// TwinCAT 3 PLC project PLC1
// ProgramVersion: 3.1.4024.12
// libraries:
//   Tc2_Standard, * (Beckhoff Automation GmbH)
//   Tc2_System, * (Beckhoff Automation GmbH)
//   Tc3_Module, * (Beckhoff Automation GmbH)
//   TcUnit,1.2.0.0,www.tcunit.org
// project tree:
//   GVLs/ GVL.TcGVL
//   / PlcTask.TcTTO
//   POUs/Casts/ CastHelper.TcPOU
//   POUs/Delegate/ Action_I_Observer_.TcPOU, Action_Person_.TcPOU, I_Action.TcIO, I_Predicate.TcIO, Predicate_Person_.TcPOU
//   POUs/ I_Equatable.TcIO, I_Observer.TcIO, Tests.TcPOU, Object.TcPOU, Person.TcPOU, PropertyObserver.TcPOU
//   POUs/List/ List.TcPOU, List_I_Observer_.TcPOU, List_Person_.TcPOU, List_Person_Test.TcPOU, List_I_Observer_Test.TcPOU

CONFIGURATION PLC1
    RESOURCE PLC ON TwinCAT3
        TASK PlcTask(INTERVAL := T#10ms, PRIORITY := 20);
        PROGRAM Tests WITH PlcTask : Tests;
    END_RESOURCE
END_CONFIGURATION

// ---- GVLs/GVL.TcGVL
{attribute 'qualified_only'}
VAR_GLOBAL
    CastHelper : CastHelper;
END_VAR
VAR_GLOBAL CONSTANT
    LIST_UPPER_BOUND : INT := 9;
END_VAR

// ---- POUs/Delegate/I_Action.TcIO
(*
Encapsulates a Perform method that has two parameters and does not return a value
*)
INTERFACE I_Action

(*
Purpose: Encapsulates several methods that can be used in the ForEach loop of a List through all elements.
Since Generic is not supported in Tc you need to implement one FB of your desired type (Action_X_) if you want to use "ForEach" method of a List that needs an Action as an input.
Because you might need several actions for different situations, it's better to write a switch-case statement and put each action in one Case instead of creating multiple FBs.
Later you can pass the CaseNumber to call your desired action.
Parameters: performCaseNumber:INT, Number to choose between actions in the method; item:POINTER TO Object, The object that is passed by the List and can be used in actions.
*)
METHOD Perform
VAR_INPUT
    performCaseNumber : INT;
END_VAR
VAR_IN_OUT
    item : POINTER TO Object;
END_VAR
END_METHOD

END_INTERFACE

// ---- POUs/Delegate/I_Predicate.TcIO
(*
Represents the Evaluate method that defines a set of criteria and determines whether the specified object meets one of those criteria
*)
INTERFACE I_Predicate

(*
Purpose: Defines a set of criteria and determines whether the specified object meets one of those criteria. 
Since Generic is not supported in Tc you need to implement one FB of your desired type (Predicated_X_) if you want to use methods of a List that need Predicate as an input.
Because you might need several criterias for different situations, it's better to write a switch-case statement and put each criteria in one Case instead of creating multiple FBs.
Later you can pass the CaseNumber to call your desired criteria.
Parameters: evaluateCaseNumber:INT, Number to choose between criterias in the method; item:POINTER TO Object, The object to compare against the criteria defined within one of the casees in the method.
Return: BOOL, True if item meets the criteria defined within the method, otherwise False.
*)
METHOD Evaluate : BOOL
VAR_INPUT
    evaluateCaseNumber : INT;
END_VAR
VAR_IN_OUT
    item : POINTER TO Object;
END_VAR
END_METHOD

END_INTERFACE

// ---- POUs/I_Equatable.TcIO
INTERFACE I_Equatable EXTENDS __System.IQueryInterface

METHOD Equals : BOOL
VAR_INPUT
    other : I_Equatable;
END_VAR
END_METHOD

END_INTERFACE

// ---- POUs/I_Observer.TcIO
INTERFACE I_Observer EXTENDS __SYSTEM.IQueryInterface, I_Equatable

METHOD OnError
VAR_INPUT
END_VAR
END_METHOD

METHOD OnUpdate
VAR_INPUT
END_VAR
END_METHOD

END_INTERFACE

// ---- POUs/Tests.TcPOU
PROGRAM Tests
VAR
    list_Person_Test : List_Person_Test;
    list_I_Observer_Test : List_I_Observer_Test;
END_VAR

TcUnit.RUN();

END_PROGRAM

// ---- POUs/List/List_Person_Test.TcPOU
FUNCTION_BLOCK List_Person_Test EXTENDS TcUnit.FB_TestSuite

AddItem();
AddRange();
Clear();
Contains();
Exists();
Find();
FindAll();
FindIndex();
FindLast();
FindLastIndex();
Foreach();
GetCapacity();
GetCount();
GetItem();
GetRange();
IndexOfItem();
LastIndexOfItem();
Initialize();
Insert();
InsertRange();
Remove();
RemoveAll();
RemoveAt();
RemoveRange();

METHOD AddItem
VAR
    personsList : List_Person_;
    personA : Person;
    personB : Person;
    actualIndex1 : INT;
    actualIndex2 : INT;
    j : INT;
END_VAR
TEST('AddPersonShouldReturnAddedIndex');
//Assign
//Act
actualIndex1 := personsList.AddItem(personA);
actualIndex2 := personsList.AddItem(personB);
//Assert
AssertEquals_INT(0, actualIndex1,'check add 1');
AssertEquals_INT(1, actualIndex2,'check add 2');
TEST_FINISHED();

TEST('AddToAFullListShouldReturnMinusOne');
//Assign
personsList.Clear();
FOR j:=0 TO GVL.LIST_UPPER_BOUND DO
    personsList.AddItem(personA);
END_FOR
//Act
actualIndex1 := personsList.AddItem(personB);
//Assert
AssertEquals_INT(-1, actualIndex1,'check overflow add');
TEST_FINISHED();
END_METHOD

METHOD AddRange
VAR
    personsList : List_Person_;
    personA : Person;
    personB : Person;
    personC : Person;
    personD : Person;
    personE : Person;
    personF : Person;
    personG : Person;
    validArrayPtPerson : ARRAY[0..2] OF POINTER TO Person := [ADR(personE), ADR(personF), ADR(personG)];
    unvalidArrayPtPerson : ARRAY[0..6 + 1] OF POINTER TO Person;
    actualPtPerson3 : POINTER TO Person;
    actualPtPerson4 : POINTER TO Person;
    actualPtPerson5 : POINTER TO Person;
    actualPtPerson6 : POINTER TO Person;
    expected : INT := 6;
    actual : INT;
END_VAR
//Before All
personA.SetAge(10);
personB.SetAge(11);
personC.SetAge(12);
personD.SetAge(13);
personE.SetAge(14);
personF.SetAge(15);
personG.SetAge(16);
personA.SetName('A');
personB.SetName('B');
personC.SetName('C');
personD.SetName('D');
personE.SetName('E');
personF.SetName('F');
personG.SetName('G');

TEST('AddRangeShouldPassAndReturnTheLastIndex');
//Assign
personsList.AddItem(personA);
personsList.AddItem(personB);
personsList.AddItem(personC);
personsList.AddItem(personD);
//Act
actual := personsList.AddRange(validArrayPtPerson);
actualPtPerson3 := personsList.GetItem(3);
actualPtPerson4 := personsList.GetItem(4);
actualPtPerson5 := personsList.GetItem(5);
actualPtPerson6 := personsList.GetItem(6);
//Assert
AssertEquals(expected, actual, 'check result');
AssertEquals_INT(7, personsList.GetCount(),'check list count');
AssertTrue(actualPtPerson3^.Equals(personD),'check added element 3');
AssertTrue(actualPtPerson4^.Equals(personE),'check added element 4');
AssertTrue(actualPtPerson5^.Equals(personF),'check added element 5');
AssertTrue(actualPtPerson6^.Equals(personG),'check added element 6');
TEST_FINISHED();

TEST('AddRangeShouldFailAndReturnMinusOne');
//Assign
personsList.Clear();
personsList.AddItem(personA);
personsList.AddItem(personB);
personsList.AddItem(personC);
personsList.AddItem(personD);
expected := -1;
//Act
actual := personsList.AddRange(unvalidArrayPtPerson);
//Assert
AssertEquals(expected, actual, 'check result');
AssertEquals_INT(4, personsList.GetCount(),'check list count');
TEST_FINISHED();
END_METHOD

METHOD Clear
VAR
    personsList1 : List_Person_;
    personsList2 : List_Person_;
    person : Person;
    expectedCount : INT := 0;
    actualCount : INT;
END_VAR
TEST('ClearAFilledListShouldPass');
//Assign
personsList1.AddItem(person);
//Act
personsList1.Clear();
actualCount := personsList1.GetCount();
//Assert
AssertEquals(expectedCount, actualCount,'');
TEST_FINISHED();

TEST('ClearAnEmptyListShouldPass');
//Assign
expectedCount := 0;
//Act
personsList2.Clear();
actualCount := personsList2.GetCount();
//Assert
AssertEquals(expectedCount, actualCount,'');
TEST_FINISHED();
END_METHOD

METHOD Contains
VAR
    personsList : List_Person_;
    personA : Person;
    personB : Person;
    personC : Person;
    personD : Person;
    personE : Person;
    personF : Person;
    personG : Person;
    actual : BOOL;
END_VAR
//Before All
personA.SetAge(10);
personB.SetAge(11);
personC.SetAge(12);
personD.SetAge(13);
personE.SetAge(14);
personF.SetAge(15);
personG.SetAge(16);
personA.SetName('A');
personB.SetName('B');
personC.SetName('C');
personD.SetName('D');
personE.SetName('E');
personF.SetName('F');
personG.SetName('G');
personsList.AddItem(personA);
personsList.AddItem(personB);
personsList.AddItem(personC);
personsList.AddItem(personD);
personsList.AddItem(personE);
personsList.AddItem(personF);

TEST('ContainsShouldReturnTrue');
//Assign
//Act
actual := personsList.Contains(personC);
//Assert
AssertTrue(actual,'Looking for personC');
TEST_FINISHED();

TEST('ContainsShouldReturnFalse');
//Assign
//Act
actual := personsList.Contains(personG);
//Assert
AssertFalse(actual,'Looking for personG');
TEST_FINISHED();
END_METHOD

METHOD Exists
VAR
    personsList : List_Person_;
    personA : Person;
    personB : Person;
    personC : Person;
    personD : Person;
    personE : Person;
    personF : Person;
    personG : Person;
    predicate_Person_ : Predicate_Person_;
    actual : BOOL;
END_VAR
//Before All
personA.SetAge(10);
personB.SetAge(11);
personC.SetAge(12);
personD.SetAge(13);
personE.SetAge(14);
personF.SetAge(15);
personG.SetAge(16);
personA.SetName('A');
personB.SetName('B');
personC.SetName('C');
personD.SetName('D');
personE.SetName('E');
personF.SetName('F');
personG.SetName('G');
personsList.AddItem(personA);
personsList.AddItem(personB);
personsList.AddItem(personC);
personsList.AddItem(personD);
personsList.AddItem(personE);
personsList.AddItem(personF);

TEST('ExistsShouldReturnTrue');
//Assign
//Act
actual := personsList.Exists(predicate_Person_, 2);
//Assert
AssertTrue(actual,'Looking for a person with name C');
TEST_FINISHED();

TEST('ExistsShouldReturnFalse');
//Assign
//Act
actual := personsList.Exists(predicate_Person_, 3);
//Assert
AssertFalse(actual,'Looking for a person with name G');
TEST_FINISHED();
END_METHOD

METHOD Find
VAR
    personsList : List_Person_;
    personA : Person;
    personB : Person;
    personC : Person;
    personD : Person;
    personE : Person;
    personF : Person;
    personG : Person;
    predicate_Person_ : Predicate_Person_;
    actualPtPerson : POINTER TO Person;
    nullPtPerson : POINTER TO person := 0;
END_VAR
//Before All
personA.SetAge(10);
personB.SetAge(11);
personC.SetAge(12);
personD.SetAge(13);
personE.SetAge(14);
personF.SetAge(15);
personG.SetAge(16);
personA.SetName('A');
personB.SetName('B');
personC.SetName('C');
personD.SetName('D');
personE.SetName('E');
personF.SetName('F');
personG.SetName('G');
personsList.AddItem(personA);
personsList.AddItem(personB);
personsList.AddItem(personC);
personsList.AddItem(personD);
personsList.AddItem(personE);
personsList.AddItem(personF);

TEST('FindShouldReturnAPerson');
//Assign
//Act
actualPtPerson := personsList.Find(predicate_Person_, 2);
//Assert
AssertTrue(actualPtPerson^.Equals(personC),'Get person with name C');
TEST_FINISHED();

TEST('FindShouldReturnZero');
//Assign
//Act
actualPtPerson := personsList.Find(predicate_Person_, 3);
//Assert
AssertEquals(nullPtPerson, actualPtPerson,'Get Zero when looking for person with name G');
TEST_FINISHED();
END_METHOD

METHOD FindAll
VAR
    personsList : List_Person_;
    personA : Person;
    personB : Person;
    personC : Person;
    personD : Person;
    personE : Person;
    personF : Person;
    predicate_Person_ : Predicate_Person_;
    actualPersonsList : list_Person_;
    actualCount : INT;
    expectedCount : INT := 3;
    actualPtPerson0 : POINTER TO Person;
    actualPtPerson1 : POINTER TO Person;
    actualPtPerson2 : POINTER TO Person;
    nullPtPerson : POINTER TO Person := 0;
END_VAR
//Before All
personA.SetAge(10);
personB.SetAge(11);
personC.SetAge(12);
personD.SetAge(13);
personE.SetAge(14);
personF.SetAge(15);
personsList.AddItem(personA);
personsList.AddItem(personB);
personsList.AddItem(personC);
personsList.AddItem(personD);
personsList.AddItem(personE);
personsList.AddItem(personF);

TEST('FindAllShouldReturnAProperList');
//Assign
//Act
actualPersonsList := personsList.FindAll(predicate_Person_, 1); //Get people younger than 13
actualCount := actualPersonsList.GetCount();
actualPtPerson0 := actualPersonsList.GetItem(0);
actualPtPerson1 := actualPersonsList.GetItem(1);
actualPtPerson2 := actualPersonsList.GetItem(2);
//Assert
AssertEquals(expectedCount, actualCount, 'Check new list count');
AssertTrue(actualPtPerson0^.Equals(personA),'First element should personA');
AssertTrue(actualPtPerson1^.Equals(personB),'First element should personB');
AssertTrue(actualPtPerson2^.Equals(personC),'First element should personC');
TEST_FINISHED();

TEST('FindAllShouldReturnAnEmptyList');
//Assign
expectedCount := 0;
//Act
actualPersonsList := personsList.FindAll(predicate_Person_, 4); //Get people older than 50
actualCount := actualPersonsList.GetCount();
actualPtPerson0 := actualPersonsList.GetItem(0);
//Assert
AssertEquals(expectedCount, actualCount, 'Check new list count');
AssertEquals(nullPtPerson, actualPtPerson0, 'Check returned list element 0');
TEST_FINISHED();
END_METHOD

METHOD FindIndex
VAR
    personsList : List_Person_;
    personA : Person;
    personB : Person;
    personC : Person;
    personD : Person;
    personE : Person;
    personF : Person;
    personG : Person;
    predicate_Person_ : Predicate_Person_;
    actualIndex : INT;
    expectedIndex : INT := 2;
END_VAR
//Before All
personA.SetAge(10);
personB.SetAge(11);
personC.SetAge(12);
personD.SetAge(13);
personE.SetAge(14);
personF.SetAge(15);
personG.SetAge(16);
personA.SetName('A');
personB.SetName('B');
personC.SetName('C');
personD.SetName('D');
personE.SetName('E');
personF.SetName('F');
personG.SetName('G');
personsList.AddItem(personA);
personsList.AddItem(personB);
personsList.AddItem(personC);
personsList.AddItem(personD);
personsList.AddItem(personE);
personsList.AddItem(personF);

TEST('FindIndexShouldReturnTheIndex');
//Assign
//Act
actualIndex := personsList.FindIndex(predicate_Person_, 2);
//Assert
AssertEquals(expectedIndex, actualIndex, 'find person with name C index');
TEST_FINISHED();

TEST('FindIndexShouldReturnMinusOne');
//Assign
expectedIndex := -1;
//Act
actualIndex := personsList.FindIndex(predicate_Person_, 3);
//Assert
AssertEquals(expectedIndex, actualIndex, 'Find person with name G index');
TEST_FINISHED();
END_METHOD

METHOD FindLast
VAR
    personsList : List_Person_;
    personA : Person;
    personB : Person;
    personC : Person;
    personC2 : Person;
    personD : Person;
    personE : Person;
    personF : Person;
    personG : Person;
    predicate_Person_ : Predicate_Person_;
    actualPtPerson : POINTER TO Person;
    nullPtPerson : POINTER TO person := 0;
END_VAR
//Before All
personA.SetAge(10);
personB.SetAge(11);
personC.SetAge(12);
personC2.SetAge(22);
personD.SetAge(13);
personE.SetAge(14);
personF.SetAge(15);
personG.SetAge(16);
personA.SetName('A');
personB.SetName('B');
personC.SetName('C');
personC2.SetName('C');
personD.SetName('D');
personE.SetName('E');
personF.SetName('F');
personG.SetName('G');
personsList.AddItem(personA);
personsList.AddItem(personB);
personsList.AddItem(personC);
personsList.AddItem(personD);
personsList.AddItem(personE);
personsList.AddItem(personC2); //Duplicated C
personsList.AddItem(personF);

TEST('FindLastShouldReturnAPerson');
//Assign
//Act
actualPtPerson := personsList.FindLast(predicate_Person_, 2);
//Assert
AssertFalse(actualPtPerson^.Equals(personC),'Not the last person with name C');
AssertTrue(actualPtPerson^.Equals(personC2),'Be the last person with name C');
TEST_FINISHED();

TEST('FindLastShouldReturnNull');
//Assign
//Act
actualPtPerson := personsList.Find(predicate_Person_, 3);
//Assert
AssertEquals(nullPtPerson, actualPtPerson,'Get Zero when looking for person with name G');
TEST_FINISHED();
END_METHOD

METHOD FindLastIndex
VAR
    personsList : List_Person_;
    personA : Person;
    personB : Person;
    personC : Person;
    personC2 : Person;
    personD : Person;
    personE : Person;
    personF : Person;
    personG : Person;
    predicate_Person_ : Predicate_Person_;
    actualIndex : INT;
    expectedIndex : INT := 5;
END_VAR
//Before All
personA.SetAge(10);
personB.SetAge(11);
personC.SetAge(12);
personC.SetAge(22);
personD.SetAge(13);
personE.SetAge(14);
personF.SetAge(15);
personG.SetAge(16);
personA.SetName('A');
personB.SetName('B');
personC.SetName('C');
personC2.SetName('C');
personD.SetName('D');
personE.SetName('E');
personF.SetName('F');
personG.SetName('G');
personsList.AddItem(personA);
personsList.AddItem(personB);
personsList.AddItem(personC);
personsList.AddItem(personD);
personsList.AddItem(personE);
personsList.AddItem(personC2);
personsList.AddItem(personF);

TEST('FindLastIndexShouldReturnTheIndex');
//Assign
//Act
actualIndex := personsList.FindLastIndex(predicate_Person_, 2);
//Assert
AssertEquals(expectedIndex, actualIndex, 'Find last person with name C index');
TEST_FINISHED();

TEST('FindLastIndexShouldReturnMinusOne');
//Assign
expectedIndex := -1;
//Act
actualIndex := personsList.FindLastIndex(predicate_Person_, 3);
//Assert
AssertEquals(expectedIndex, actualIndex, 'Find person with name G index');
TEST_FINISHED();
END_METHOD

METHOD Foreach
VAR
    personsList : List_Person_;
    personA : Person;
    personB : Person;
    personC : Person;
    personD : Person;
    personE : Person;
    personF : Person;
    personG : Person;
    action_Person_ : Action_Person_;
    actualPtPersonArray : ARRAY[0..3] OF POINTER TO Person;
    j : INT;
    expectedName : STRING := 'John';
END_VAR
TEST('ForeachShouldPass');
//Assign
personA.SetAge(10);
personB.SetAge(11);
personC.SetAge(12);
personD.SetAge(13);
personE.SetAge(14);
personF.SetAge(15);
personG.SetAge(16);
personA.SetName('A');
personB.SetName('B');
personC.SetName('C');
personD.SetName('D');
personE.SetName('E');
personF.SetName('F');
personG.SetName('G');
personsList.AddItem(personA);
personsList.AddItem(personB);
personsList.AddItem(personC);
personsList.AddItem(personD);
//Act
personsList.Foreach(action_Person_, 2);
FOR j:=0 TO 3 DO
    actualPtPersonArray[j] := personsList.GetItem(j);
END_FOR
//Assert
AssertEquals_STRING(expectedName, actualPtPersonArray[0]^.GetName(),'element 0 shuold be named John');
AssertEquals_STRING(expectedName, actualPtPersonArray[1]^.GetName(),'element 0 shuold be named John');
AssertEquals_STRING(expectedName, actualPtPersonArray[2]^.GetName(),'element 0 shuold be named John');
AssertEquals_STRING(expectedName, actualPtPersonArray[3]^.GetName(),'element 0 shuold be named John');
TEST_FINISHED();
END_METHOD

METHOD GetCapacity
VAR
    personsList : List_Person_;
    person : Person;
    expectedCapacity : INT := GVL.LIST_UPPER_BOUND + 1;
    actualCapacity : INT;
END_VAR
TEST('GetCapacityShouldPass');
//Act
actualCapacity := personsList.GetCapacity();
//Assert
AssertEquals_INT(expectedCapacity, actualCapacity,'Get capacity at the begining');
TEST_FINISHED();

TEST('GetCapacityShouldPassWithSameValue');
//Assign
personsList.AddItem(person);
//Act
actualCapacity := personsList.GetCapacity();
//Assert
AssertEquals(expectedCapacity, actualCapacity,'Get capacity after adding a person');
TEST_FINISHED();
END_METHOD

METHOD GetCount
VAR
    personsList : List_Person_;
    person : Person;
    expectedCount : INT := 0;
    actualCount : INT;
END_VAR
TEST('GetCountShouldReturnZero');
//Act
actualCount := personsList.GetCount();
//Assert
AssertEquals_INT(expectedCount, actualCount,'Get count at the begining');
TEST_FINISHED();

TEST('GetCountShouldReturnOne');
//Assign
personsList.AddItem(person);
expectedCount := 1;
//Act
actualCount := personsList.GetCount();
//Assert
AssertEquals(expectedCount, actualCount,'Get count after adding a person');
TEST_FINISHED();
END_METHOD

METHOD GetItem
VAR
    personsList : List_Person_;
    personA : Person;
    personB : Person;
    actualPtPerson : POINTER TO Person;
END_VAR
//Before All
personA.SetAge(10);
personB.SetAge(11);
personA.SetName('A');
personB.SetName('B');
personsList.AddItem(personA);
personsList.AddItem(personB);

TEST('GetPersonShouldPass');
//Assign
//Act
actualPtPerson := personsList.GetItem(1);
//Assert
AssertEquals_INT(11, actualPtPerson^.GetAge(),'check age');
AssertTrue(actualPtPerson^.Equals(personB),'check Equality');
TEST_FINISHED();

TEST('GetShouldBeByReference');
//Assign
//Act
actualPtPerson := personsList.GetItem(1);
personB.SetAge(20);
actualPtPerson^.GetAge();
//Assert
AssertEquals_INT(20, actualPtPerson^.GetAge(),'');
TEST_FINISHED();
END_METHOD

METHOD GetRange
VAR
    personsList : List_Person_;
    personA : Person;
    personB : Person;
    personC : Person;
    personD : Person;
    personE : Person;
    personF : Person;
    personG : Person;
    actualPersonsList : list_Person_;
    actualCount : INT;
    expectedCount : INT := 3;
    actualPtPerson0 : POINTER TO Person;
    actualPtPerson1 : POINTER TO Person;
    actualPtPerson2 : POINTER TO Person;
END_VAR
//Before All
personA.SetAge(10);
personB.SetAge(11);
personC.SetAge(12);
personD.SetAge(13);
personE.SetAge(14);
personF.SetAge(15);
personG.SetAge(16);
personsList.AddItem(personA);
personsList.AddItem(personB);
personsList.AddItem(personC);
personsList.AddItem(personD);
personsList.AddItem(personE);
personsList.AddItem(personF);

TEST('GetRangeShouldReturnList');
//Assign
//Act
actualPersonsList := personsList.GetRange(1, expectedCount);
actualCount := actualPersonsList.GetCount();
actualPtPerson0 := actualPersonsList.GetItem(0);
actualPtPerson1 := actualPersonsList.GetItem(1);
actualPtPerson2 := actualPersonsList.GetItem(2);
//Assert
AssertEquals(expectedCount, actualCount, 'Check new list count');
AssertTrue(actualPtPerson0^.Equals(personB),'First element should personB');
AssertTrue(actualPtPerson1^.Equals(personC),'First element should personC');
AssertTrue(actualPtPerson2^.Equals(personD),'First element should personD');
TEST_FINISHED();

TEST('GetRangeShouldReturnListTillLastElement');
//Assign
//Act
actualPersonsList := personsList.GetRange(1, 1000);
actualCount := actualPersonsList.GetCount();
//Assert
expectedCount := 5;
AssertEquals(expectedCount, actualCount, 'Check new list count for GetRange 1000');
TEST_FINISHED();

TEST('GetRangeShouldReturnEmptyList');
//Assign
//Act
actualPersonsList := personsList.GetRange(-5, 1);
actualCount := actualPersonsList.GetCount();
//Assert
expectedCount := 0;
AssertEquals(expectedCount, actualCount, 'Check new list count for GetRange starting -5');
TEST_FINISHED();
END_METHOD

METHOD IndexOfItem
VAR
    personsList : List_Person_;
    personA : Person;
    personB : Person;
    personC : Person;
    personD : Person;
    personE : Person;
    personF : Person;
    personG : Person;
    actualIndex : INT;
    expectedIndex : INT := 3;
END_VAR
//Before All
personA.SetAge(10);
personB.SetAge(11);
personC.SetAge(12);
personD.SetAge(13);
personE.SetAge(14);
personF.SetAge(15);
personG.SetAge(16);
personA.SetName('A');
personB.SetName('B');
personC.SetName('C');
personD.SetName('D');
personE.SetName('E');
personF.SetName('F');
personG.SetName('G');
personsList.AddItem(personA);
personsList.AddItem(personB);
personsList.AddItem(personC);
personsList.AddItem(personD);
personsList.AddItem(personE);
personsList.AddItem(personF);

TEST('IndexOfItemShouldReturnTheIndex');
//Assign
//Act
actualIndex := personsList.IndexOfItem(personD);
//Assert
AssertEquals(expectedIndex, actualIndex, 'return the index of personD');
TEST_FINISHED();

TEST('IndexOfItemShouldReturnMinusOne');
//Assign
//Act
actualIndex := personsList.IndexOfItem(personG);
//Assert
expectedIndex := -1;
AssertEquals(expectedIndex, actualIndex, 'return the index of personG');
TEST_FINISHED();
END_METHOD

METHOD Initialize
VAR
    personsList : List_Person_;
    personA : Person;
    personB : Person;
    personC : Person;
    validArrayPtPerson : ARRAY[0..2] OF POINTER TO Person := [ADR(personA), ADR(personB), ADR(personC)];
    unvalidArrayPtPerson : ARRAY[0..GVL.LIST_UPPER_BOUND + 1] OF POINTER TO Person;
    actualPtPerson0 : POINTER TO Person;
    actualPtPerson1 : POINTER TO Person;
    actualPtPerson2 : POINTER TO Person;
    expected : INT := 2;
    actual : INT;
END_VAR
//Before All
personA.SetAge(10);
personB.SetAge(11);
personC.SetAge(12);
personA.SetName('A');
personB.SetName('B');
personC.SetName('C');

TEST('InitializeShouldPassAndReturnTheLastIndex');
//Assign
//Act
actual := personsList.Initialize(validArrayPtPerson);
actualPtPerson0 := personsList.GetItem(0);
actualPtPerson1 := personsList.GetItem(1);
actualPtPerson2 := personsList.GetItem(2);
//Assert
AssertEquals(expected, actual, 'check result');
AssertEquals_INT(3, personsList.GetCount(),'check list count');
AssertTrue(actualPtPerson0^.Equals(personA),'check added element 0');
AssertTrue(actualPtPerson1^.Equals(personB),'check added element 1');
AssertTrue(actualPtPerson2^.Equals(personC),'check added element 2');
TEST_FINISHED();

TEST('InitializeShouldFailAndReturnMinusOne');
//Assign
personsList.Clear();
expected := -1;
//Act
actual := personsList.Initialize(unvalidArrayPtPerson);
//Assert
AssertEquals(expected, actual, 'check result');
AssertEquals_INT(0, personsList.GetCount(),'check list count');
TEST_FINISHED();
END_METHOD

METHOD Insert
VAR
    personsList : List_Person_;
    personA : Person;
    personB : Person;
    personC : Person;
    personD : Person;
    actualPtPerson1 : POINTER TO Person;
    actualPtPerson2 : POINTER TO Person;
    actualPtPerson3 : POINTER TO Person;
    expected : INT := 2;
    actual : INT;
END_VAR
//Before All
personA.SetAge(10);
personB.SetAge(11);
personC.SetAge(12);
personD.SetAge(13);
personA.SetName('A');
personB.SetName('B');
personC.SetName('C');
personD.SetName('D');

TEST('InsertShouldPassAndReturnTheLastIndex');
//Assign
personsList.AddItem(personA);
personsList.AddItem(personB);
personsList.AddItem(personC);
//Act
actual := personsList.Insert(2, personD);
actualPtPerson1 := personsList.GetItem(1);
actualPtPerson2 := personsList.GetItem(2);
actualPtPerson3 := personsList.GetItem(3);
//Assert
AssertEquals(expected, actual, 'check result');
AssertEquals_INT(4, personsList.GetCount(),'check list count');
AssertTrue(actualPtPerson1^.Equals(personB),'check added element 1');
AssertTrue(actualPtPerson2^.Equals(personD),'check added element 2');
AssertTrue(actualPtPerson3^.Equals(personC),'check added element 3');
TEST_FINISHED();

TEST('InsertShouldPassEvenByIndexHigherThanListCurrentLastIndexAndReturnTheLastIndex');
//Assign
personsList.Clear();
personsList.AddItem(personA);
personsList.AddItem(personB);
personsList.AddItem(personC);
expected := 3;
//Act
actual := personsList.Insert(7, personD);
actualPtPerson1 := personsList.GetItem(1);
actualPtPerson2 := personsList.GetItem(2);
actualPtPerson3 := personsList.GetItem(3);
//Assert
AssertEquals(expected, actual, 'check result');
AssertEquals_INT(4, personsList.GetCount(),'check list count');
AssertTrue(actualPtPerson1^.Equals(personB),'check added element 1');
AssertTrue(actualPtPerson2^.Equals(personC),'check added element 2');
AssertTrue(actualPtPerson3^.Equals(personD),'check added element 3');
TEST_FINISHED();

TEST('InsertShouldPassEvenByIndexHigherThanListUpperBoundAndReturnTheLastIndex');
//Assign
personsList.Clear();
personsList.AddItem(personA);
personsList.AddItem(personB);
personsList.AddItem(personC);
expected := 3;
//Act
actual := personsList.Insert(GVL.LIST_UPPER_BOUND + 1, personD);
actualPtPerson1 := personsList.GetItem(1);
actualPtPerson2 := personsList.GetItem(2);
actualPtPerson3 := personsList.GetItem(3);
//Assert
AssertEquals(expected, actual, 'check result');
AssertEquals_INT(4, personsList.GetCount(),'check list count');
AssertTrue(actualPtPerson1^.Equals(personB),'check added element 1');
AssertTrue(actualPtPerson2^.Equals(personC),'check added element 2');
AssertTrue(actualPtPerson3^.Equals(personD),'check added element 3');
TEST_FINISHED();

TEST('InsertShouldFailByMinusIndexAndReturnMinusOne');
//Assign
personsList.Clear();
personsList.AddItem(personA);
personsList.AddItem(personB);
personsList.AddItem(personC);
expected := -1;
//Act
actual := personsList.Insert(-1, personD);
//Assert
AssertEquals(expected, actual, 'check result');
AssertEquals_INT(3, personsList.GetCount(),'check list count');
TEST_FINISHED();
END_METHOD

METHOD InsertRange
VAR
    personsList : List_Person_;
    personA : Person;
    personB : Person;
    personC : Person;
    personD : Person;
    personE : Person;
    personF : Person;
    personG : Person;
    validArrayPtPerson : ARRAY[0..2] OF POINTER TO Person := [ADR(personE), ADR(personF), ADR(personG)];
    unvalidArrayPtPerson : ARRAY[0..6 + 1] OF POINTER TO Person;
    actualPtPerson1 : POINTER TO Person;
    actualPtPerson2 : POINTER TO Person;
    actualPtPerson3 : POINTER TO Person;
    actualPtPerson4 : POINTER TO Person;
    actualPtPerson5 : POINTER TO Person;
    actualPtPerson6 : POINTER TO Person;
    actualPtPerson7 : POINTER TO Person;
    expected : INT := 4;
    actual : INT;
END_VAR
//Before All
personA.SetAge(10);
personB.SetAge(11);
personC.SetAge(12);
personD.SetAge(13);
personE.SetAge(14);
personF.SetAge(15);
personG.SetAge(16);
personA.SetName('A');
personB.SetName('B');
personC.SetName('C');
personD.SetName('D');
personE.SetName('E');
personF.SetName('F');
personG.SetName('G');

TEST('InsertRangeShouldPassAndReturnTheLastIndex');
//Assign
personsList.AddItem(personA);
personsList.AddItem(personB);
personsList.AddItem(personC);
personsList.AddItem(personD);
//Act
actual := personsList.InsertRange(2, validArrayPtPerson);
actualPtPerson1 := personsList.GetItem(1);
actualPtPerson2 := personsList.GetItem(2);
actualPtPerson3 := personsList.GetItem(3);
actualPtPerson4 := personsList.GetItem(4);
actualPtPerson5 := personsList.GetItem(5);
//Assert
AssertEquals(expected, actual, 'check result');
AssertEquals_INT(7, personsList.GetCount(),'check list count');
AssertTrue(actualPtPerson1^.Equals(personB),'check added element 1');
AssertTrue(actualPtPerson2^.Equals(personE),'check added element 2');
AssertTrue(actualPtPerson3^.Equals(personF),'check added element 3');
AssertTrue(actualPtPerson4^.Equals(personG),'check added element 4');
AssertTrue(actualPtPerson5^.Equals(personC),'check added element 5');
TEST_FINISHED();

TEST('InsertRangeShouldPassEvenByIndexHigherThanListCurrentLastIndexAndReturnTheLastIndex');
//Assign
personsList.Clear();
personsList.AddItem(personA);
personsList.AddItem(personB);
personsList.AddItem(personC);
personsList.AddItem(personD);
expected := 6;
//Act
actual := personsList.InsertRange(7, validArrayPtPerson);
actualPtPerson3 := personsList.GetItem(3);
actualPtPerson4 := personsList.GetItem(4);
actualPtPerson5 := personsList.GetItem(5);
actualPtPerson6 := personsList.GetItem(6);
//Assert
AssertEquals(expected, actual, 'check result');
AssertEquals_INT(7, personsList.GetCount(),'check list count');
AssertTrue(actualPtPerson3^.Equals(personD),'check added element 3');
AssertTrue(actualPtPerson4^.Equals(personE),'check added element 4');
AssertTrue(actualPtPerson5^.Equals(personF),'check added element 5');
AssertTrue(actualPtPerson6^.Equals(personG),'check added element 6');
TEST_FINISHED();

TEST('InsertRangeShouldPassEvenByIndexHigherThanListUpperBoundAndReturnTheLastIndex');
//Assign
personsList.Clear();
personsList.AddItem(personA);
personsList.AddItem(personB);
personsList.AddItem(personC);
personsList.AddItem(personD);
expected := 6;
//Act
actual := personsList.InsertRange(7, validArrayPtPerson);
actualPtPerson3 := personsList.GetItem(3);
actualPtPerson4 := personsList.GetItem(4);
actualPtPerson5 := personsList.GetItem(5);
actualPtPerson6 := personsList.GetItem(6);
//Assert
AssertEquals(expected, actual, 'check result');
AssertEquals_INT(7, personsList.GetCount(),'check list count');
AssertTrue(actualPtPerson3^.Equals(personD),'check added element 3');
AssertTrue(actualPtPerson4^.Equals(personE),'check added element 4');
AssertTrue(actualPtPerson5^.Equals(personF),'check added element 5');
AssertTrue(actualPtPerson6^.Equals(personG),'check added element 6');
TEST_FINISHED();

TEST('InsertRangeShouldFailByMinusIndexAndReturnMinusOne');
//Assign
personsList.Clear();
personsList.AddItem(personA);
personsList.AddItem(personB);
personsList.AddItem(personC);
personsList.AddItem(personD);
expected := -1;
//Act
actual := personsList.InsertRange(-1, validArrayPtPerson);
//Assert
AssertEquals(expected, actual, 'check result');
AssertEquals_INT(4, personsList.GetCount(),'check list count');
TEST_FINISHED();

TEST('InsertRangeShouldFailByLongArrayLengthAndReturnMinusOne');
//Assign
personsList.Clear();
personsList.AddItem(personA);
personsList.AddItem(personB);
personsList.AddItem(personC);
personsList.AddItem(personD);
expected := -1;
//Act
actual := personsList.InsertRange(2, unvalidArrayPtPerson);
//Assert
AssertEquals(expected, actual, 'check result');
AssertEquals_INT(4, personsList.GetCount(),'check list count');
TEST_FINISHED();
END_METHOD

METHOD LastIndexOfItem
VAR
    personsList : List_Person_;
    personA : Person;
    personB : Person;
    personC : Person;
    personD : Person;
    personE : Person;
    personF : Person;
    personG : Person;
    actualIndex : INT;
    expectedIndex : INT := 5;
END_VAR
//Before All
personA.SetAge(10);
personB.SetAge(11);
personC.SetAge(12);
personD.SetAge(13);
personE.SetAge(14);
personF.SetAge(15);
personG.SetAge(16);
personA.SetName('A');
personB.SetName('B');
personC.SetName('C');
personD.SetName('D');
personE.SetName('E');
personF.SetName('F');
personG.SetName('G');
personsList.AddItem(personA);
personsList.AddItem(personB);
personsList.AddItem(personC);
personsList.AddItem(personD);
personsList.AddItem(personE);
personsList.AddItem(personD);
personsList.AddItem(personF);

TEST('LastIndexOfItemShouldReturnTheIndex');
//Assign
//Act
actualIndex := personsList.LastIndexOfItem(personD);
//Assert
AssertEquals(expectedIndex, actualIndex, 'return the last index of personD');
TEST_FINISHED();

TEST('LastIndexOfItemShouldReturnMinusOne');
//Assign
//Act
actualIndex := personsList.LastIndexOfItem(personG);
//Assert
expectedIndex := -1;
AssertEquals(expectedIndex, actualIndex, 'return the last index of personG');
TEST_FINISHED();
END_METHOD

METHOD Remove
VAR
    personsList : List_Person_;
    personA : Person;
    personB : Person;
    personC : Person;
    personD : Person;
    expectedCount : INT := 3;
    actualPtPerson1 : POINTER TO Person;
    actualPtPerson2 : POINTER TO Person;
    actualCount : INT;
    actual : BOOL;
END_VAR
//Before All
personA.SetAge(10);
personB.SetAge(11);
personC.SetAge(12);
personD.SetAge(13);
personA.SetName('A');
personB.SetName('B');
personC.SetName('C');
personD.SetName('D');
personsList.AddItem(personA);
personsList.AddItem(personB);
personsList.AddItem(personC);
personsList.AddItem(personD);

TEST('RemoveShouldPassAndReturnTrue');
//Assign
//Act
actual := personsList.Remove(personC);
actualCount := personsList.GetCount();
actualPtPerson1 := personsList.GetItem(1);
actualPtPerson2 := personsList.GetItem(2);
//Assert
AssertTrue(actual,'check result of remove');
AssertEquals(expectedCount, actualCount,'check list count');
AssertTrue(actualPtPerson1^.Equals(personB),'check list element 1');
AssertTrue(actualPtPerson2^.Equals(personD),'check list element 2');
TEST_FINISHED();

TEST('RemoveShouldFailAndReturnFalse');
//Assign
//Act
actual := personsList.Remove(personC);
actualCount := personsList.GetCount();
actualPtPerson1 := personsList.GetItem(1);
actualPtPerson2 := personsList.GetItem(2);
//Assert
AssertFalse(actual,'check result of remove');
AssertEquals(expectedCount, actualCount,'check list count');
AssertTrue(actualPtPerson1^.Equals(personB),'check list element 1');
AssertTrue(actualPtPerson2^.Equals(personD),'check list element 2');
TEST_FINISHED();
END_METHOD

METHOD RemoveAll
VAR
    personsList : List_Person_;
    personA : Person;
    personB : Person;
    personC : Person;
    personD : Person;
    personE : Person;
    personF : Person;
    personG : Person;
    predicate_Person_ : Predicate_Person_;
    actual : INT;
    expected : INT := 3;
    actualCount : INT;
    expectedCount : INT := 4;
    actualPtPerson0 : POINTER TO Person;
    actualPtPerson1 : POINTER TO Person;
    actualPtPerson2 : POINTER TO Person;
    actualPtPerson3 : POINTER TO Person;
    actualPtPerson4 : POINTER TO Person;
    actualPtPerson5 : POINTER TO Person;
    actualPtPerson6 : POINTER TO Person;
END_VAR
//Before All
personA.SetAge(10);
personB.SetAge(11);
personC.SetAge(12);
personD.SetAge(13);
personE.SetAge(14);
personF.SetAge(15);
personG.SetAge(16);

TEST('RemoveAllShouldReturnAProperList');
//Assign
personsList.AddItem(personA);
personsList.AddItem(personB);
personsList.AddItem(personC);
personsList.AddItem(personD);
personsList.AddItem(personE);
personsList.AddItem(personF);
personsList.AddItem(personG);
//Act
actual := personsList.RemoveAll(predicate_Person_, 1); //Remove people younger than 13
actualCount := personsList.GetCount();
actualPtPerson0 := personsList.GetItem(0);
actualPtPerson1 := personsList.GetItem(1);
actualPtPerson2 := personsList.GetItem(2);
actualPtPerson3 := personsList.GetItem(3);
//Assert
AssertEquals(expected, actual, 'check result');
AssertEquals(expectedCount, actualCount, 'check list count');
AssertTrue(actualPtPerson0^.Equals(personD),'check returned list element 0');
AssertTrue(actualPtPerson1^.Equals(personE),'check returned list element 1');
AssertTrue(actualPtPerson2^.Equals(personF),'check returned list element 2');
AssertTrue(actualPtPerson3^.Equals(personG),'check returned list element 3');
TEST_FINISHED();

TEST('RemoveAllShouldReturnTheOriginalListUntouched');
//Assign
personsList.Clear();
personsList.AddItem(personA);
personsList.AddItem(personB);
personsList.AddItem(personC);
personsList.AddItem(personD);
personsList.AddItem(personE);
personsList.AddItem(personF);
personsList.AddItem(personG);
expected := 0;
expectedCount := 7;
//Act
actual := personsList.RemoveAll(predicate_Person_, 4); //Remove people older than 50
actualCount := personsList.GetCount();
actualPtPerson0 := personsList.GetItem(0);
actualPtPerson1 := personsList.GetItem(1);
actualPtPerson2 := personsList.GetItem(2);
actualPtPerson3 := personsList.GetItem(3);
actualPtPerson4 := personsList.GetItem(4);
actualPtPerson5 := personsList.GetItem(5);
actualPtPerson6 := personsList.GetItem(6);
//Assert
AssertEquals(expected, actual, 'check result');
AssertEquals(expectedCount, actualCount, 'check list count');
AssertTrue(actualPtPerson0^.Equals(personA),'check returned list element 0');
AssertTrue(actualPtPerson1^.Equals(personB),'check returned list element 1');
AssertTrue(actualPtPerson2^.Equals(personC),'check returned list element 2');
AssertTrue(actualPtPerson3^.Equals(personD),'check returned list element 3');
AssertTrue(actualPtPerson4^.Equals(personE),'check returned list element 4');
AssertTrue(actualPtPerson5^.Equals(personF),'check returned list element 5');
AssertTrue(actualPtPerson6^.Equals(personG),'check returned list element 6');
TEST_FINISHED();
END_METHOD

METHOD RemoveAt
VAR
    personsList : List_Person_;
    personA : Person;
    personB : Person;
    personC : Person;
    personD : Person;
    actualPtPersonArray : ARRAY[0..3] OF POINTER TO Person;
    expectedCount : INT := 3;
    actualCount : INT;
    actual : BOOL;
    j : INT;
END_VAR
//Before All
personA.SetAge(10);
personB.SetAge(11);
personC.SetAge(12);
personD.SetAge(13);
personA.SetName('A');
personB.SetName('B');
personC.SetName('C');
personD.SetName('D');

TEST('RemoveAtShouldPass');
//Assign
personsList.Clear();
personsList.AddItem(personA);
personsList.AddItem(personB);
personsList.AddItem(personC);
personsList.AddItem(personD);
//Act
actual := personsList.RemoveAt(2);
actualCount := personsList.GetCount();
FOR j:=0 TO 3 DO
    actualPtPersonArray[j] := personsList.GetItem(j);
END_FOR
//Assert
AssertTrue(actual,'check result of remove');
AssertEquals(expectedCount, actualCount,'check list count');
AssertTrue(actualPtPersonArray[0]^.Equals(personA),'check element 0');
AssertTrue(actualPtPersonArray[1]^.Equals(personB),'check element 1');
AssertTrue(actualPtPersonArray[2]^.Equals(personD),'check element 2');
TEST_FINISHED();

TEST('RemoveAtMinusIndexShouldFail');
//Assign
personsList.Clear();
personsList.AddItem(personA);
personsList.AddItem(personB);
personsList.AddItem(personC);
personsList.AddItem(personD);
expectedCount := 4;
//Act
actual := personsList.RemoveAt(-1);
actualCount := personsList.GetCount();
FOR j:=0 TO 3 DO
    actualPtPersonArray[j] := personsList.GetItem(j);
END_FOR
//Assert
AssertFalse(actual,'check result of remove');
AssertEquals(expectedCount, actualCount,'check list count');
AssertTrue(actualPtPersonArray[0]^.Equals(personA),'check element 0');
AssertTrue(actualPtPersonArray[1]^.Equals(personB),'check element 1');
AssertTrue(actualPtPersonArray[2]^.Equals(personC),'check element 2');
AssertTrue(actualPtPersonArray[3]^.Equals(personD),'check element 3');
TEST_FINISHED();

TEST('RemoveAtIndexGreaterThanLastIndexShouldFail');
//Assign
personsList.Clear();
personsList.AddItem(personA);
personsList.AddItem(personB);
personsList.AddItem(personC);
personsList.AddItem(personD);
expectedCount := 4;
//Act
actualCount := personsList.GetCount();
actual := personsList.RemoveAt(actualCount);
actualCount := personsList.GetCount();
FOR j:=0 TO 3 DO
    actualPtPersonArray[j] := personsList.GetItem(j);
END_FOR
//Assert
AssertFalse(actual,'check result of remove');
AssertEquals(expectedCount, actualCount,'check list count');
AssertTrue(actualPtPersonArray[0]^.Equals(personA),'check element 0');
AssertTrue(actualPtPersonArray[1]^.Equals(personB),'check element 1');
AssertTrue(actualPtPersonArray[2]^.Equals(personC),'check element 2');
AssertTrue(actualPtPersonArray[3]^.Equals(personD),'check element 3');
TEST_FINISHED();
END_METHOD

METHOD RemoveRange
VAR
    personsList : List_Person_;
    personA : Person;
    personB : Person;
    personC : Person;
    personD : Person;
    personE : Person;
    personF : Person;
    personG : Person;
    actualPtPersonArray : ARRAY[0..3] OF POINTER TO Person;
    expectedCount : INT := 7 - 3;
    actualCount : INT;
    actual : BOOL;
    j : INT;
END_VAR
//Before All
personA.SetAge(10);
personB.SetAge(11);
personC.SetAge(12);
personD.SetAge(13);
personE.SetAge(14);
personF.SetAge(15);
personG.SetAge(16);
personA.SetName('A');
personB.SetName('B');
personC.SetName('C');
personD.SetName('D');
personE.SetName('E');
personF.SetName('F');
personG.SetName('G');

TEST('RemoveRangeShouldPass');
//Assign
personsList.AddItem(personA);
personsList.AddItem(personB);
personsList.AddItem(personC);
personsList.AddItem(personD);
personsList.AddItem(personE);
personsList.AddItem(personF);
personsList.AddItem(personG);
//Act
actual := personsList.RemoveRange(2,3);
actualCount := personsList.GetCount();
FOR j:=0 TO 3 DO
    actualPtPersonArray[j] := personsList.GetItem(j);
END_FOR
//Assert
AssertTrue(actual,'check result of removeRange');
AssertEquals(expectedCount, actualCount,'check list count');
AssertTrue(actualPtPersonArray[0]^.Equals(personA),'check element 0');
AssertTrue(actualPtPersonArray[1]^.Equals(personB),'check element 1');
AssertTrue(actualPtPersonArray[2]^.Equals(personF),'check element 2');
AssertTrue(actualPtPersonArray[3]^.Equals(personG),'check element 3');
TEST_FINISHED();

TEST('RemoveRangeWithRangeLongerThanCountShouldPass');
//Assign
personsList.Clear();
personsList.AddItem(personA);
personsList.AddItem(personB);
personsList.AddItem(personC);
personsList.AddItem(personD);
personsList.AddItem(personE);
personsList.AddItem(personF);
personsList.AddItem(personG);
expectedCount := 4;
//Act
actual := personsList.RemoveRange(4,10);
actualCount := personsList.GetCount();
FOR j:=0 TO 3 DO
    actualPtPersonArray[j] := personsList.GetItem(j);
END_FOR
//Assert
AssertTrue(actual,'check result of removeRange');
AssertEquals(expectedCount, actualCount,'check list count');
AssertTrue(actualPtPersonArray[0]^.Equals(personA),'check element 0');
AssertTrue(actualPtPersonArray[1]^.Equals(personB),'check element 1');
AssertTrue(actualPtPersonArray[2]^.Equals(personC),'check element 2');
AssertTrue(actualPtPersonArray[3]^.Equals(personD),'check element 3');
TEST_FINISHED();

TEST('RemoveRangeWithMinusIndexShouldFail');
//Assign
personsList.Clear();
personsList.AddItem(personA);
personsList.AddItem(personB);
personsList.AddItem(personC);
personsList.AddItem(personD);
personsList.AddItem(personE);
personsList.AddItem(personF);
personsList.AddItem(personG);
expectedCount := 7;
//Act
actual := personsList.RemoveRange(-1,3);
actualCount := personsList.GetCount();
FOR j:=0 TO 3 DO
    actualPtPersonArray[j] := personsList.GetItem(j);
END_FOR
//Assert
AssertFalse(actual,'check result of removeRange');
AssertEquals(expectedCount, actualCount,'check list count');
AssertTrue(actualPtPersonArray[0]^.Equals(personA),'check element 0');
AssertTrue(actualPtPersonArray[1]^.Equals(personB),'check element 1');
AssertTrue(actualPtPersonArray[2]^.Equals(personC),'check element 2');
AssertTrue(actualPtPersonArray[3]^.Equals(personD),'check element 3');
TEST_FINISHED();

TEST('RemoveRangeWithIndexGreaterThanLastIndexShouldFail');
//Assign
personsList.Clear();
personsList.AddItem(personA);
personsList.AddItem(personB);
personsList.AddItem(personC);
personsList.AddItem(personD);
personsList.AddItem(personE);
personsList.AddItem(personF);
personsList.AddItem(personG);
expectedCount := 7;
//Act
actualCount := personsList.GetCount();
actual := personsList.RemoveRange(actualCount,3);
actualCount := personsList.GetCount();
FOR j:=0 TO 3 DO
    actualPtPersonArray[j] := personsList.GetItem(j);
END_FOR
//Assert
AssertFalse(actual,'check result of removeRange');
AssertEquals(expectedCount, actualCount,'check list count');
AssertTrue(actualPtPersonArray[0]^.Equals(personA),'check element 0');
AssertTrue(actualPtPersonArray[1]^.Equals(personB),'check element 1');
AssertTrue(actualPtPersonArray[2]^.Equals(personC),'check element 2');
AssertTrue(actualPtPersonArray[3]^.Equals(personD),'check element 3');
TEST_FINISHED();
END_METHOD

END_FUNCTION_BLOCK

// ---- POUs/List/List_Person_.TcPOU
(*
Sample List which has all available functionalities.
For instance this is a list of type Person (C# eq: List<Person>).
To have any desired type (!!!Not Interface!!!) make a copy of this FB and change Person to your type in all methods
*)
FUNCTION_BLOCK FINAL List_Person_ EXTENDS List

(*
Purpose: Adds an item to the end of the List
Parameters: item:{X Extends Object}, The object to be added to the end of the List
Return: INT, The zero-based index of added object if item is added, otherwise -1
*)
METHOD PUBLIC AddItem : INT
VAR_IN_OUT
    item : Person;
END_VAR
AddItem := SUPER^._addItem(item);
END_METHOD

(*
Purpose: Adds elements of the specified array to the end of the List
Parameters: items:ARRAY[*] OF POINTER TO {X Extends Object}, The array whose elements should be added to the end of the List
Return: INT, The zero-based index of the last added object if items are added, otherwise -1
*)
METHOD PUBLIC AddRange : INT
VAR_IN_OUT
    items : ARRAY[*] OF POINTER TO Person;
END_VAR
AddRange := SUPER^._addRange(items);
END_METHOD

(*
Purpose: Determines whether an element is in the List
Parameters: item:{X Extends Object}, The object to locate in the List
Return: BOOL, True if item is found in the List, otherwise False
*)
METHOD PUBLIC Contains : BOOL
VAR_IN_OUT
    item: Person;
END_VAR
Contains := SUPER^._contains(item);
END_METHOD

(*
Purpose: Determines whether the List contains elements that match the condition defined by the specified predicate
Parameters: predicate:{Predicate_X_ Implements IPredicate}, The Predicate delegate that defines the conditions of the elements to search for; evaluateCaseNumber:INT, Number that specifies which condition to evaluate
Return: BOOL, True if the List contains one or more elements that match the condition defined by the specified predicate, otherwise False
*)
METHOD PUBLIC Exists : BOOL
VAR_INPUT
    predicate: Predicate_Person_;
    evaluateCaseNumber : INT;
END_VAR
Exists := SUPER^._exists(predicate, evaluateCaseNumber);
END_METHOD

(*
Purpose: Searches for an element that matches the conditions defined by the specified predicate, and returns the first occurrence within the entire List
Parameters: predicate:{Predicate_X_ Implements IPredicate}, The Predicate delegate that defines the conditions of the elements to search for; evaluateCaseNumber:INT, Number that specifies which condition to evaluate
Return: POINTER TO {X Extends Object}, The address of the first element that matches the conditions defined by the specified predicate if found, otherwise 0
*)
METHOD Find : POINTER TO Person
VAR_INPUT
    predicate: Predicate_Person_;
    evaluateCaseNumber : INT;
END_VAR
Find := SUPER^._find(predicate, evaluateCaseNumber);
END_METHOD

(*
Purpose: Retrieves all the elements that match the conditions defined by the specified predicate
Parameters: predicate:{Predicate_X_ Implements IPredicate}, The Predicate delegate that defines the conditions of the elements to search for; evaluateCaseNumber:INT, Number that specifies which condition to evaluate
Return: {List_X_ Extends List}, A List containing all the elements that match the conditions defined by the specified predicate if found, otherwise an empty List
*)
METHOD FindAll: List_Person_
VAR_INPUT
    predicate: Predicate_Person_;
    evaluateCaseNumber : INT;
END_VAR
FindAll := GVL.CastHelper.ListToList_Person_(SUPER^._findAll(predicate, evaluateCaseNumber));
END_METHOD

(*
Purpose: Searches for an element that matches the conditions defined by a specified predicate and returns the zero-based index of the first occurrence within the List
Parameters: predicate:{Predicate_X_ Implements IPredicate}, The Predicate delegate that defines the conditions of the elements to search for; evaluateCaseNumber:INT, Number that specifies which condition to evaluate
Return: INT, The zero-based index of the first occurrence of an element that matches the conditions defined by match if found, otherwise -1.
*)
METHOD FindIndex : INT
VAR_INPUT
    predicate: Predicate_Person_;
    evaluateCaseNumber : INT;
END_VAR
FindIndex := SUPER^._findIndex(predicate, evaluateCaseNumber);
END_METHOD

(*
Purpose: Searches for an element that matches the conditions defined by the specified predicate, and returns the last occurrence within the entire List
Parameters: predicate:{X Implements IPredicate}, The Predicate delegate that defines the conditions of the elements to search for; evaluateCaseNumber:INT, Number that specifies which condition to evaluate
Return: POINTER TO {X Extends Object}, The address of the last element that matches the conditions defined by the specified predicate if found, otherwise 0
*)
METHOD FindLast : POINTER TO Person
VAR_INPUT
    predicate: Predicate_Person_;
    evaluateCaseNumber : INT;
END_VAR
FindLast := SUPER^._findLast(predicate, evaluateCaseNumber);
END_METHOD

(*
Purpose: Searches for an element that matches the conditions defined by a specified predicate and returns the zero-based index of the last occurrence within the List
Parameters: predicate:{X Implements IPredicate}, The Predicate delegate that defines the conditions of the elements to search for; evaluateCaseNumber:INT, Number that specifies which condition to evaluate
Return: INT, The zero-based index of the last occurrence of an element that matches the conditions defined by match if found, otherwise -1.
*)
METHOD FindLastIndex : INT
VAR_INPUT
    predicate: Predicate_Person_;
    evaluateCaseNumber : INT;
END_VAR
FindLastIndex := SUPER^._findLastIndex(predicate, evaluateCaseNumber);
END_METHOD

(*
Purpose: Performs the specified action on each element of the List
Parameters: _action:{Action_X_ Implements IAction}, The Action delegate to perform on each element of the List; performCaseNumber:INT, Number that specifies which action to perform
Return: BOOL, True if the action is performed on all elements, otherwise False
*)
METHOD Foreach: BOOL
VAR_INPUT
    _action : I_Action;
    performCaseNumber : INT;
END_VAR
Foreach := SUPER^._forEach(_action, performCaseNumber);
END_METHOD

(*
Purpose: Gets the element at the specified index
Parameters: index:INT, The zero-based index of the element to get
Return: POINTER TO {X Extends Object}, The element at the specified index
*)
METHOD PUBLIC GetItem : POINTER TO Person
VAR_INPUT
    index : INT;
END_VAR
GetItem := SUPER^.GetItemAsIEquatable(index);
END_METHOD

(*
Purpose: Creates a shallow copy of a range of elements in the source List
Parameters: index:INT, The zero-based List index at which the range starts; count:INT, The number of elements in the range
Return: {List_X_ Extends List}, A shallow copy of a range of elements in the source List
*)
METHOD PUBLIC GetRange: List_Person_
VAR_INPUT
    index : INT;
    count : INT;
END_VAR
GetRange := GVL.CastHelper.ListToList_Person_(SUPER^._getRange(index, count));
END_METHOD

(*
Purpose: Returns the zero-based index of the first occurrence in the List
Parameters: item:{X Extends Object}, The object to locate in the List
Return: INT, The zero-based index of the first occurrence of item in the List if found, otherwise -1
*)
METHOD PUBLIC IndexOfItem : INT
VAR_IN_OUT
    item: Person;
END_VAR
IndexOfItem := SUPER^._indexOf(item);
END_METHOD

(*
Purpose: Initializes the List by copying the specified array
Parameters: items:ARRAY[*] OF POINTER TO {X Extends Object}, The array whose elements are copied to the new list
Return: INT, The zero-based index of the last copied element if input array length is less or equal to length of the list, otherwise -1
*)
METHOD PUBLIC Initialize : INT
VAR_IN_OUT
    items : ARRAY[*] OF POINTER TO Person;
END_VAR
Initialize := _initialize(items);
END_METHOD

(*
Purpose: Inserts an item at the specified index
Parameters: index:INT ,The zero-based index at which the new object should be inserted; item:{X Extends Object}, The object to insert
Return: INT, The zero-based index of the inserted object if inserted, otherwise -1
*)
METHOD PUBLIC Insert : INT
VAR_INPUT
    index : INT;
END_VAR
VAR_IN_OUT
    item : Person;
END_VAR
Insert := SUPER^._insert(index, item);
END_METHOD

(*
Purpose: Inserts elements of the specified array at the specified index
Parameters: index:INT ,The zero-based index at which the new elements should be inserted; items:ARRAY[*] OF POINTER TO {X Extends Object}, The array whose elements should be inserted into the List
Return: INT, The zero-based index of the last inserted object if input array length is less or equal to remaining capacity of the list, otherwise -1
*)
METHOD PUBLIC InsertRange : INT
VAR_INPUT
    index : INT;
END_VAR
VAR_IN_OUT
    items : ARRAY[*] OF POINTER TO Person;
END_VAR
InsertRange := SUPER^._insertRange(index, items);
END_METHOD

(*
Purpose: Returns the zero-based index of the last occurrence in the List
Parameters: item:{X Extends Object}, The object to locate in the List
Return: INT, The zero-based index of the last occurrence of item in the List if found, otherwise -1
*)
METHOD PUBLIC LastIndexOfItem : INT
VAR_IN_OUT
    item: Person;
END_VAR
LastIndexOfItem := SUPER^._lastIndexOf(item);
END_METHOD

(*
Purpose: Removes the address of the first occurrence of a specific object from the List
Parameters: item:{X Extends Object}, The object to remove from the List
Return: BOOL, True if item is successfully removed, otherwise False
*)
METHOD PUBLIC Remove : BOOL
VAR_IN_OUT
    item: Person;
END_VAR
Remove := SUPER^._remove(item);
END_METHOD

(*
Purpose: Removes all the elements that match the conditions defined by the specified predicate
Parameters: predicate:{Predicate_X_ Implements IPredicate}, The Predicate delegate that defines the conditions of the elements to search for; evaluateCaseNumber:INT, Number that specifies which condition to evaluate
Return: INT, The number of elements removed from the List
*)
METHOD RemoveAll : INT
VAR_INPUT
    predicate: Predicate_Person_;
    evaluateCaseNumber : INT;
END_VAR
RemoveAll := SUPER^._removeAll(predicate, evaluateCaseNumber);
END_METHOD

(*
Purpose: Copies the elements of the List to a new array
Return: ARRAY[0..GVL.LIST_UPPER_BOUND] OF POINTER TO {X Extends Object}, An array containing copies of the elements of the List as {X Extends Object}
*)
METHOD PUBLIC ToArray : ARRAY[0..GVL.LIST_UPPER_BOUND] OF POINTER TO Person
VAR
    i : INT;
    arrayOfIEquatable : ARRAY[0..GVL.LIST_UPPER_BOUND] OF POINTER TO I_Equatable;
    _result : ARRAY[0..GVL.LIST_UPPER_BOUND] OF POINTER TO Person;
END_VAR
arrayOfIEquatable := SUPER^._toArray();
FOR i:=0 TO GetCount() - 1 DO
    _result[i] := arrayOfIEquatable[i];
END_FOR

ToArray := _result;
END_METHOD

END_FUNCTION_BLOCK

// ---- POUs/List/List.TcPOU
(*
Base List which includes core and generic functionality of a list.
To have a list of any desired type (X) a new FB that Extends this FB should be created which can implement any desired Protected methods of this FB.
*)
FUNCTION_BLOCK List
VAR_INPUT
END_VAR
VAR_OUTPUT
END_VAR
VAR
    _internalArray : ARRAY [0..GVL.LIST_UPPER_BOUND] OF LWORD;
    _count : INT := 0;
END_VAR

(*
Purpose: Adds the address of an Object to the end of the List
Parameters: item:Object, The object to be added to the end of the List
Return: INT, The zero-based index of added object if item is added, otherwise -1
*)
METHOD PROTECTED _addItem : INT
VAR_IN_OUT
    item : Object;
END_VAR
VAR
    _result : INT := -1;
END_VAR
IF GetCount() <= GVL.LIST_UPPER_BOUND THEN
    _internalArray[_count] := ADR(item);
    _result := _count;
    _count := _count + 1;
END_IF
_addItem := _result;
END_METHOD

(*
Purpose: Adds the address of the elements of the specified array to the end of the List
Parameters: items:ARRAY[*] OF POINTER TO Object, The array whose elements should be added to the end of the List
Return: INT, The zero-based index of the last added object if items are added, otherwise -1
*)
METHOD PROTECTED _addRange : INT
VAR_IN_OUT
    items : ARRAY[*] OF POINTER TO Object;
END_VAR
VAR
    _result : INT := -1;
    _lowerBound : DINT;
    _upperBound : DINT;
    _itemsLength : DINT;
    i : DINT;
END_VAR
_lowerBound := LOWER_BOUND(items,1);
_upperBound := UPPER_BOUND(items,1);
_itemsLength := _upperBound - _lowerBound + 1;
IF _itemsLength <= GetCapacity() - GetCount() THEN
    FOR i := _lowerBound TO _upperBound DO
        _addItem(items[i]^);
	END_FOR
    _result := DINT_TO_INT(GetCount() - 1);
END_IF

_addRange := _result;
END_METHOD

(*
Purpose: Determines whether an element is in the List
Parameters: item:Object, The object to locate in the List
Return: BOOL, True if item is found in the List, otherwise False
*)
METHOD PROTECTED _contains : BOOL
VAR_IN_OUT
    item : Object;
END_VAR
VAR
    i : INT;
    _lastIndex : INT;
    _currentItem : POINTER TO Object;
    _result : BOOL := False;
END_VAR
IF GetCount() > 0 THEN
    _lastIndex := GetCount() - 1;
    FOR i:=0 TO _lastIndex DO
        _currentItem := GetItemAsIEquatable(i);
        IF _currentItem^.Equals(item) THEN
            _result := TRUE;
            EXIT;
        END_IF
    END_FOR
END_IF

_contains := _result;
END_METHOD

(*
Purpose: Determines whether the List contains elements that match the condition defined by the specified predicate
Parameters: predicate:IPredicate, The Predicate delegate that defines the conditions of the elements to search for; evaluateCaseNumber:INT, Number that specifies which condition to evaluate
Return: BOOL, True if the List contains one or more elements that match the condition defined by the specified predicate, otherwise False
*)
METHOD PROTECTED _exists : BOOL
VAR_INPUT
    predicate : I_Predicate;
    evaluateCaseNumber : INT;
END_VAR
VAR
    i : INT;
    _lastIndex : INT;
    _currentItem : POINTER TO Object;
    _result : BOOL := FALSE;
END_VAR
IF GetCount() > 0 THEN
    _lastIndex := GetCount() - 1;
    FOR i:=0 TO _lastIndex DO
        _currentItem := GetItemAsIEquatable(i);
        IF predicate.Evaluate(evaluateCaseNumber, _currentItem) THEN
            _result := TRUE;
            EXIT;
        END_IF
    END_FOR
END_IF

_exists := _result;
END_METHOD

(*
Purpose: Searches for an element that matches the conditions defined by the specified predicate, and returns the first occurrence within the entire List
Parameters: predicate:IPredicate, The Predicate delegate that defines the conditions of the elements to search for; evaluateCaseNumber:INT, Number that specifies which condition to evaluate
Return: POINTER TO Object, The address of the first element that matches the conditions defined by the specified predicate if found, otherwise 0
*)
METHOD PROTECTED _find : POINTER TO Object
VAR_INPUT
    predicate : I_Predicate;
    evaluateCaseNumber : INT;
END_VAR
VAR
    i : INT;
    _lastIndex : INT;
    _currentItem : POINTER TO Object;
    _result : POINTER TO Object := 0;
END_VAR
IF GetCount() > 0 THEN
    _lastIndex := GetCount() - 1;
    FOR i:=0 TO _lastIndex DO
        _currentItem := GetItemAsIEquatable(i);
        IF predicate.Evaluate(evaluateCaseNumber, _currentItem) THEN
            _result := _currentItem;
            EXIT;
        END_IF
    END_FOR
END_IF

_find := _result;
END_METHOD

(*
Purpose: Retrieves all the elements that match the conditions defined by the specified predicate
Parameters: predicate:IPredicate, The Predicate delegate that defines the conditions of the elements to search for; evaluateCaseNumber:INT, Number that specifies which condition to evaluate
Return: List, A List containing all the elements that match the conditions defined by the specified predicate if found, otherwise an empty List
*)
METHOD PROTECTED _findAll : List
VAR_INPUT
    predicate : I_Predicate;
    evaluateCaseNumber : INT;
END_VAR
VAR
    i : INT;
    _lastIndex : INT;
    _currentItem : POINTER TO Object;
    _result : List;
END_VAR
IF GetCount() > 0 THEN
    _lastIndex := GetCount() - 1;
    FOR i:=0 TO _lastIndex DO
        _currentItem := GetItemAsIEquatable(i);
        IF predicate.Evaluate(evaluateCaseNumber, _currentItem) THEN
            _result._addItem(_currentItem^);
        END_IF
    END_FOR
END_IF

_findAll := _result;
END_METHOD

(*
Purpose: Searches for an element that matches the conditions defined by a specified predicate and returns the zero-based index of the first occurrence within the List
Parameters: predicate:IPredicate, The Predicate delegate that defines the conditions of the elements to search for; evaluateCaseNumber:INT, Number that specifies which condition to evaluate
Return: INT, The zero-based index of the first occurrence of an element that matches the conditions defined by match if found, otherwise -1.
*)
METHOD PROTECTED _findIndex : INT
VAR_INPUT
    predicate : I_Predicate;
    evaluateCaseNumber : INT;
END_VAR
VAR
    i : INT;
    _lastIndex : INT;
    _currentItem : POINTER TO Object;
    _result : INT := -1;
END_VAR
IF GetCount() > 0 THEN
    _lastIndex := GetCount() - 1;
    FOR i:=0 TO _lastIndex DO
        _currentItem := GetItemAsIEquatable(i);
        IF predicate.Evaluate(evaluateCaseNumber, _currentItem) THEN
            _result := i;
            EXIT;
        END_IF
    END_FOR
END_IF

_findIndex := _result;
END_METHOD

(*
Purpose: Searches for an element that matches the conditions defined by the specified predicate, and returns the last occurrence within the entire List
Parameters: predicate:IPredicate, The Predicate delegate that defines the conditions of the elements to search for; evaluateCaseNumber:INT, Number that specifies which condition to evaluate
Return: POINTER TO Object, The address of the last element that matches the conditions defined by the specified predicate if found, otherwise 0
*)
METHOD PROTECTED _findLast : POINTER TO Object
VAR_INPUT
    predicate : I_Predicate;
    evaluateCaseNumber : INT;
END_VAR
VAR
    i : INT;
    _lastIndex : INT;
    _currentItem : POINTER TO Object;
    _result : POINTER TO Object := 0;
END_VAR
IF GetCount() > 0 THEN
    _lastIndex := GetCount() - 1;
    FOR i:=0 TO _lastIndex DO
        _currentItem := GetItemAsIEquatable(_lastIndex - i);
        IF predicate.Evaluate(evaluateCaseNumber, _currentItem) THEN
            _result := _currentItem;
            EXIT;
        END_IF
    END_FOR
END_IF

_findLast := _result;
END_METHOD

(*
Purpose: Searches for an element that matches the conditions defined by a specified predicate and returns the zero-based index of the last occurrence within the List
Parameters: predicate:IPredicate, The Predicate delegate that defines the conditions of the elements to search for; evaluateCaseNumber:INT, Number that specifies which condition to evaluate
Return: INT, The zero-based index of the last occurrence of an element that matches the conditions defined by match if found, otherwise -1.
*)
METHOD PROTECTED _findLastIndex : INT
VAR_INPUT
    predicate : I_Predicate;
    evaluateCaseNumber : INT;
END_VAR
VAR
    i : INT;
    _lastIndex : INT;
    _currentItem : POINTER TO Object;
    _result : INT := -1;
END_VAR
IF GetCount() > 0 THEN
    _lastIndex := GetCount() - 1;
    FOR i:=0 TO _lastIndex DO
        _currentItem := GetItemAsIEquatable(_lastIndex - i);
        IF predicate.Evaluate(evaluateCaseNumber, _currentItem) THEN
            _result := _lastIndex - i;
            EXIT;
        END_IF
    END_FOR
END_IF

_findLastIndex := _result;
END_METHOD

(*
Purpose: Performs the specified action on each element of the List
Parameters: _action:IAction, The Action delegate to perform on each element of the List; performCaseNumber:INT, Number that specifies which action to perform
Return: BOOL, True if the action is performed on all elements, otherwise False
*)
METHOD PROTECTED _forEach : BOOL
VAR_INPUT
    _action : I_Action;
    performCaseNumber : INT;
END_VAR
VAR
    i : INT;
    _lastIndex : INT;
    _currentItem : POINTER TO Object;
    ex : __SYSTEM.ExceptionCode;
    _result : BOOL;
END_VAR
//__TRY  (*not supported on x64 systems*)
    IF GetCount() > 0 THEN
        _lastIndex := GetCount() - 1;
        FOR i:=0 TO _lastIndex DO
            _currentItem := GetItemAsIEquatable(i);
            _action.Perform(performCaseNumber, _currentItem);
        END_FOR
        _result := TRUE;
    END_IF
//__CATCH(ex)
//    _result := FALSE;
//__ENDTRY

_forEach := _result;
END_METHOD

(*
Purpose: Creates a shallow copy of a range of elements in the source List
Parameters: index:INT, The zero-based List index at which the range starts; count:INT, The number of elements in the range
Return: List, A shallow copy of a range of elements in the source List
*)
METHOD PROTECTED _getRange : List
VAR_INPUT
    index : INT;
    count : INT;
END_VAR
VAR
    i : INT;
    _lastIndex : INT;
    _lastIndexToGet : INT;
    _currentItem : POINTER TO Object;
    _result : List;
END_VAR
IF GetCount() > 0 AND_THEN index >= 0 AND_THEN count > 0 THEN
    _lastIndex := GetCount() - 1;
    IF index <= _lastIndex THEN
        _lastIndexToGet := index + count - 1;
        IF _lastIndexToGet > _lastIndex THEN
            _lastIndexToGet := _lastIndex;
        END_IF
        FOR i := index TO _lastIndexToGet DO
            _currentItem := GetItemAsIEquatable(i);
            _result._addItem(_currentItem^);
        END_FOR
    END_IF
END_IF

_getRange := _result;
END_METHOD

(*
Purpose: Returns the zero-based index of the first occurrence in the List
Parameters: item:Object, The object to locate in the List
Return: INT, The zero-based index of the first occurrence of item in the List if found, otherwise -1
*)
METHOD PROTECTED _indexOf : INT
VAR_IN_OUT
    item : Object;
END_VAR
VAR
    i : INT;
    _lastIndex : INT;
    _currentItem : POINTER TO Object;
    _result : INT := -1;
END_VAR
IF GetCount() > 0 THEN
    _lastIndex := GetCount() - 1;
    FOR i:=0 TO _lastIndex DO
        _currentItem := GetItemAsIEquatable(i);
        IF _currentItem^.Equals(item) THEN
            _result := i;
            EXIT;
        END_IF
    END_FOR
END_IF

_indexOf := _result;
END_METHOD

(*
Purpose: Initializes the List by copying the specified array
Parameters: items:ARRAY[*] OF POINTER TO Object, The array whose elements are copied to the new list
Return: INT, The zero-based index of the last copied element if input array length is less or equal to length of the list, otherwise -1
*)
METHOD PROTECTED _initialize : INT
VAR_IN_OUT
    items : ARRAY[*] OF POINTER TO Object;
END_VAR
VAR
    _result : INT := -1;
    _lowerBound : DINT;
    _upperBound : DINT;
    _itemsLength : DINT;
    i : DINT;
END_VAR
_lowerBound := LOWER_BOUND(items,1);
_upperBound := UPPER_BOUND(items,1);
_itemsLength := _upperBound - _lowerBound + 1;
IF _itemsLength <= GetCapacity() THEN
    Clear();
    _result := _addRange(items);
END_IF

_initialize := _result;
END_METHOD

(*
Purpose: Inserts the address of the Object at the specified index
Parameters: index:INT ,The zero-based index at which the new object should be inserted; item:Object, The object to insert
Return: INT, The zero-based index of the inserted object if inserted, otherwise -1
*)
METHOD PROTECTED _insert : INT
VAR_INPUT
    index : INT;
END_VAR
VAR_IN_OUT
    item : Object;
END_VAR
VAR
    i : INT;
    _result : INT := -1;
    count : INT;
END_VAR
count := GetCount();
IF count <= GVL.LIST_UPPER_BOUND AND index >= 0 THEN
    IF index >= count THEN
        _result := _addItem(item);
    ELSE
        FOR i:=0 TO count - index - 1 DO
            _internalArray[count - i] := _internalArray[count - i - 1];
        END_FOR
        _internalArray[index] := ADR(item);
        _count := _count + 1;
        _result := index;
    END_IF
END_IF

_insert := _result;
END_METHOD

(*
Purpose: Inserts the address of the elements of the specified array at the specified index
Parameters: index:INT ,The zero-based index at which the new elements should be inserted; items:ARRAY[*] OF POINTER TO Object, The array whose elements should be inserted into the List
Return: INT, The zero-based index of the last inserted object if input array length is less or equal to remaining capacity of the list, otherwise -1
*)
METHOD PROTECTED _insertRange : INT
VAR_INPUT
    index : INT;
END_VAR
VAR_IN_OUT
    items : ARRAY[*] OF POINTER TO Object;
END_VAR
VAR
    _result : INT := -1;
    _lowerBound : DINT;
    _upperBound : DINT;
    _itemsLength : DINT;
    i : DINT;
    j : INT := 0;
END_VAR
IF index >= 0 THEN
    IF index < GetCount() THEN
        _lowerBound := LOWER_BOUND(items,1);
        _upperBound := UPPER_BOUND(items,1);
        _itemsLength := _upperBound - _lowerBound + 1;
        IF _itemsLength <= GetCapacity() - GetCount() THEN
            FOR i := _lowerBound TO _upperBound DO
                _result := _insert(index + j, items[i]^);
                j := j + 1;
            END_FOR
        END_IF
    ELSE
        _result := _addRange(items);
	END_IF
END_IF

_insertRange := _result;
END_METHOD

(*
Purpose: Returns the zero-based index of the last occurrence in the List
Parameters: item:Object, The object to locate in the List
Return: INT, The zero-based index of the last occurrence of item in the List if found, otherwise -1
*)
METHOD PROTECTED _lastIndexOf : INT
VAR_IN_OUT
    item : Object;
END_VAR
VAR
    i : INT;
    _lastIndex : INT;
    _currentItem : POINTER TO Object;
    _result : INT := -1;
END_VAR
IF GetCount() > 0 THEN
    _lastIndex := GetCount() - 1;
    FOR i:=0 TO _lastIndex DO
        _currentItem := GetItemAsIEquatable(_lastIndex - i);
        IF _currentItem^.Equals(item) THEN
            _result := _lastIndex - i;
            EXIT;
        END_IF
    END_FOR
END_IF

_lastIndexOf := _result;
END_METHOD

(*
Purpose: Removes the address of the first occurrence of a specific object from the List
Parameters: item:Object, The object to remove from the List
Return: BOOL, True if item is successfully removed, otherwise False
*)
METHOD PROTECTED _remove : BOOL
VAR_IN_OUT
    item : Object;
END_VAR
VAR
    i : INT;
    _lastIndex : INT;
    _currentItem : POINTER TO Object;
    _result : BOOL := FALSE;
END_VAR
IF GetCount() > 0 THEN
    _lastIndex := GetCount() - 1;
    FOR i:=0 TO _lastIndex DO
        _currentItem := GetItemAsIEquatable(i);
        IF _currentItem^.Equals(item) THEN
            _result := RemoveAt(i);
            EXIT;
        END_IF
    END_FOR
END_IF

_remove := _result;
END_METHOD

(*
Purpose: Removes all the elements that match the conditions defined by the specified predicate
Parameters: predicate:IPredicate, The Predicate delegate that defines the conditions of the elements to search for; evaluateCaseNumber:INT, Number that specifies which condition to evaluate
Return: INT, The number of elements removed from the List
*)
METHOD PROTECTED _removeAll : INT
VAR_INPUT
    predicate : I_Predicate;
    evaluateCaseNumber : INT;
END_VAR
VAR
    i : INT;
    _lastIndex : INT;
    _currentItem : POINTER TO Object;
    _result : INT;
END_VAR
IF GetCount() > 0 THEN
    _lastIndex := GetCount() - 1;
    FOR i:=0 TO _lastIndex DO
        _currentItem := GetItemAsIEquatable(i);
        IF predicate.Evaluate(evaluateCaseNumber, _currentItem) THEN
            _remove(_currentItem^);
            i := i - 1;
            _lastIndex := _lastIndex - 1;
            _result := _result + 1;
        END_IF
    END_FOR
END_IF

_removeAll := _result;
END_METHOD

(*
Purpose: Copies the elements of the List to a new array
Return: ARRAY[0..GVL.LIST_UPPER_BOUND] OF POINTER TO IEquatable, An array containing copies of the elements of the List as IEquatable
*)
METHOD PROTECTED _toArray : ARRAY[0..GVL.LIST_UPPER_BOUND] OF POINTER TO I_Equatable
VAR
    i : INT;
    count : INT;
    _result : ARRAY[0..GVL.LIST_UPPER_BOUND] OF POINTER TO I_Equatable;
END_VAR
count := GetCount();
IF count > 0 THEN
    FOR i:=0 TO count - 1 DO
        _result[i] := GVL.CastHelper.AddressToI_Equatable(_internalArray[i]);
    END_FOR
END_IF

_toArray := _result;
END_METHOD

(*
Purpose: Removes all elements from the List
*)
METHOD PUBLIC Clear
VAR
    i : INT;
END_VAR
IF GetCount() > 0 THEN
    FOR i:= 0 TO GetCount()-1 DO
        _internalArray[i] := 0;
    END_FOR
    _count := 0;
END_IF
END_METHOD

(*
Purpose: Gets the total number of elements the internal array can hold regardless of added elements
Return: INT, The number of elements that the List can contain
*)
METHOD PUBLIC GetCapacity : INT
GetCapacity := GVL.LIST_UPPER_BOUND + 1;
END_METHOD

(*
Purpose: Gets the number of elements contained in the List
Return: INT, The number of elements contained in the List
*)
METHOD PUBLIC GetCount : INT
GetCount := _count;
END_METHOD

(*
Purpose: Gets the element at the specified index
Parameters: index:INT, The zero-based index of the element to get
Return: POINTER TO IEquatable, The element at the specified index
*)
METHOD PUBLIC GetItemAsIEquatable : POINTER TO I_Equatable
VAR_INPUT
    index : INT;
END_VAR
IF GetCount() = 0 OR_ELSE index < 0 OR_ELSE index >= _count THEN
    GetItemAsIEquatable := 0;
ELSE
    GetItemAsIEquatable := GVL.CastHelper.AddressToI_Equatable(_internalArray[index]);
END_IF
END_METHOD

(*
Purpose: Removes the element at the specified index of the List
Parameters: index:INT, The zero-based index of the element to remove
Return: BOOL, True if the element is removed, otherwise False
*)
METHOD PUBLIC RemoveAt : BOOL
VAR_INPUT
    index : INT;
END_VAR
VAR
    i : INT;
    _lastIndex : INT;
    _result : BOOL := FALSE;
END_VAR
IF GetCount() > 0 AND_THEN index >= 0 THEN
    _lastIndex := GetCount() - 1;
    IF index <= _lastIndex THEN
        FOR i := index TO _lastIndex - 1 DO
            _internalArray[i] := _internalArray[i + 1];
        END_FOR
        _internalArray[_lastIndex] := 0;
        _count := GetCount() - 1;
        _result := TRUE;
    END_IF
END_IF

RemoveAt := _result;
END_METHOD

(*
Purpose: Removes a range of elements from the List
Parameters: index:INT, The zero-based starting index of the range of elements to remove; count:INT, The number of elements to remove
Return: BOOL, True if the last element is removed, otherwise False
*)
METHOD PUBLIC RemoveRange : BOOL
VAR_INPUT
    index : INT;
    count : INT;
END_VAR
VAR
    i : INT;
    _lastIndex : INT;
    _lastIndexToRemove : INT;
    _result : BOOL := FALSE;
END_VAR
IF GetCount() > 0 AND_THEN index >= 0 AND_THEN count > 0 THEN
    _lastIndex := GetCount() - 1;
    IF index <= _lastIndex THEN
        _lastIndexToRemove := index + count - 1;
        IF _lastIndexToRemove > _lastIndex THEN
            _lastIndexToRemove := _lastIndex;
        END_IF
        FOR i := index TO _lastIndexToRemove DO
            _result := RemoveAt(index);
        END_FOR
    END_IF
END_IF

RemoveRange := _result;
END_METHOD

END_FUNCTION_BLOCK

// ---- POUs/Object.TcPOU
FUNCTION_BLOCK Object IMPLEMENTS I_Equatable
VAR_INPUT
END_VAR
VAR_OUTPUT
END_VAR
VAR
END_VAR

METHOD Equals : BOOL
VAR_INPUT
    other : I_Equatable;
END_VAR
Equals := false;
END_METHOD

END_FUNCTION_BLOCK

// ---- POUs/Casts/CastHelper.TcPOU
(*
To pass objects between List (base) and List_X_ (derived) we need to cast types. Since these castings are used in several methods, they are all gathered here is this FB.
AddressToI_Equatable is general for all lists.
I_EquatableToX, ListToList_X & ObjectToX (X here indicates your desired object type) should be implemented foreach type that you want to create a list of.
In this project for instance I created Person FB, then a List_Person_ and I_EquatableToPerson, ListToList_Person & ObjectToPerson. You can copy these methods and rename any "Person" to the name of your FB.
*)
FUNCTION_BLOCK FINAL CastHelper
VAR_INPUT
END_VAR
VAR_OUTPUT
END_VAR
VAR
END_VAR

METHOD AddressToI_Equatable : POINTER TO I_Equatable
VAR_IN_OUT
	item : LWORD;
END_VAR
VAR
    _pointerToCastedItem : POINTER TO I_Equatable;
    _pointerToPointer : POINTER TO LWORD := ADR(_pointerToCastedItem);
END_VAR
_pointerToPointer^ := item;
AddressToI_Equatable := _pointerToCastedItem;
END_METHOD

METHOD I_EquatableToPerson : POINTER TO Person
VAR_IN_OUT
	item : I_Equatable;
END_VAR
VAR
    _pointerToCastedItem : POINTER TO Person;
END_VAR
__QUERYPOINTER(item, _pointerToCastedItem);
I_EquatableToPerson := _pointerToCastedItem;
END_METHOD

METHOD I_EquatableToPropertyObserver : POINTER TO PropertyObserver
VAR_IN_OUT
	item : I_Equatable;
END_VAR
VAR
    _pointerToCastedItem : POINTER TO PropertyObserver;
END_VAR
__QUERYPOINTER(item, _pointerToCastedItem);
I_EquatableToPropertyObserver := _pointerToCastedItem;
END_METHOD

METHOD PUBLIC ListToList_Person_ : List_Person_
VAR_INPUT
    list : List;
END_VAR
VAR
    i : INT;
    lastIndex : INT;
    _currentItem : POINTER TO Object;
    _result : List_Person_;
END_VAR
IF list.GetCount() > 0 THEN
    lastIndex := list.GetCount()-1;
    IF lastIndex >= 0 THEN
        FOR i:=0 TO lastIndex DO
            _currentItem := list.GetItemAsIEquatable(i);
            _result.AddItem(GVL.CastHelper.ObjectToPerson(_currentItem)^);
        END_FOR
    END_IF
END_IF

ListToList_Person_ := _result;
END_METHOD

METHOD ObjectToPerson : POINTER TO Person
VAR_IN_OUT
	item : POINTER TO Object;
END_VAR
VAR
    _pointerToCastedItem : POINTER TO Person;
    _pointerToPointer : POINTER TO LWORD := ADR(_pointerToCastedItem);
END_VAR
_pointerToPointer^ := item;
ObjectToPerson := _pointerToCastedItem;
END_METHOD

END_FUNCTION_BLOCK

// ---- POUs/Person.TcPOU
FUNCTION_BLOCK Person Extends Object
VAR_INPUT
END_VAR
VAR_OUTPUT
END_VAR
VAR
    _age : INT;
    _name : STRING;
END_VAR

METHOD Equals : BOOL
VAR_INPUT
    other : I_Equatable;
END_VAR
IF GetAge() = GVL.CastHelper.I_EquatableToPerson(other)^.GetAge() THEN
    Equals := TRUE;
ELSE
    Equals := FALSE;
END_IF
END_METHOD

METHOD GetAge : int
VAR_INPUT
END_VAR
GetAge := _age;
END_METHOD

METHOD PUBLIC GetName : STRING
GetName := _name;
END_METHOD

METHOD SetAge : int
VAR_INPUT
    age : int;
END_VAR
_age := age;
SetAge := _age;
END_METHOD

METHOD PUBLIC SetName : STRING
VAR_INPUT
    name : STRING;
END_VAR
_name := name;
SetName := _name;
END_METHOD

END_FUNCTION_BLOCK

// ---- POUs/PropertyObserver.TcPOU
FUNCTION_BLOCK PropertyObserver EXTENDS Object IMPLEMENTS I_Observer
VAR_INPUT
END_VAR
VAR_OUTPUT
END_VAR
VAR
    _name : STRING;
    _counter : INT;
END_VAR

METHOD Equals : BOOL
VAR_INPUT
    other : I_Equatable;
END_VAR
IF GetCounter() = GVL.CastHelper.I_EquatableToPropertyObserver(other)^.GetCounter() THEN
    Equals := TRUE;
ELSE
    Equals := FALSE;
END_IF
END_METHOD

METHOD GetCounter : INT
VAR_INPUT
END_VAR
GetCounter := _counter;
END_METHOD

METHOD OnError
_counter := _counter - 1;
END_METHOD

METHOD OnUpdate
_counter := _counter + 1;
END_METHOD

METHOD SetCounter
VAR_INPUT
    counter : INT;
END_VAR
_counter := counter;
END_METHOD

END_FUNCTION_BLOCK

// ---- POUs/Delegate/Predicate_Person_.TcPOU
(*
You can use this FB as a template for your Predicates. Rename "Person" to your "typeName" and add your criterias.
*)
FUNCTION_BLOCK FINAL Predicate_Person_ IMPLEMENTS I_Predicate

(*
Purpose: Defines a set of criteria and determines whether the specified object meets one of those criteria. 
Since Generic is not supported in Tc you need to implement one FB of your desired type (Predicated_X_) if you want to use methods of a List that need Predicate as an input.
Because you might need several criterias for different situations, it's better to write a switch-case statement and put each criteria in one Case instead of creating multiple FBs.
Later you can pass the CaseNumber to call your desired criteria.
Parameters: evaluateCaseNumber:INT, Number to choose between criterias in the method; item:POINTER TO Object, The object to compare against the criteria defined within one of the casees in the method.
Return: BOOL, True if item meets the criteria defined within the method, otherwise False.
*)
METHOD Evaluate : BOOL
VAR_INPUT
    evaluateCaseNumber : INT;
END_VAR
VAR_IN_OUT
	item : POINTER TO Object;
END_VAR
CASE evaluateCaseNumber OF
    1 :
    IF GVL.CastHelper.ObjectToPerson(item)^.GetAge() < 13 THEN
        Evaluate := TRUE;
    ELSE
        Evaluate := FALSE;
    END_IF
    2 :
    IF GVL.CastHelper.ObjectToPerson(item)^.GetName() = 'C' THEN
        Evaluate := TRUE;
    ELSE
        Evaluate := FALSE;
    END_IF
    3 :
    IF GVL.CastHelper.ObjectToPerson(item)^.GetName() = 'G' THEN
        Evaluate := TRUE;
    ELSE
        Evaluate := FALSE;
    END_IF
    4 :
    IF GVL.CastHelper.ObjectToPerson(item)^.GetAge() > 50 THEN
        Evaluate := TRUE;
    ELSE
        Evaluate := FALSE;
    END_IF
ELSE
    Evaluate := FALSE;
END_CASE
END_METHOD

END_FUNCTION_BLOCK

// ---- POUs/Delegate/Action_Person_.TcPOU
FUNCTION_BLOCK FINAL Action_Person_ IMPLEMENTS I_Action

(*
Purpose: Encapsulates several methods that can be used in the ForEach loop of a List through all elements.
Since Generic is not supported in Tc you need to implement one FB of your desired type (Action_X_) if you want to use "ForEach" method of a List that needs an Action as an input.
Because you might need several actions for different situations, it's better to write a switch-case statement and put each action in one Case instead of creating multiple FBs.
Later you can pass the CaseNumber to call your desired action.
Parameters: performCaseNumber:INT, Number to choose between actions in the method; item:POINTER TO Object, The object that is passed by the List and can be used in actions.
*)
METHOD Perform
VAR_INPUT
    performCaseNumber : INT;
END_VAR
VAR_IN_OUT
	item : POINTER TO Object;
END_VAR
CASE performCaseNumber OF
    1 :
    GVL.CastHelper.ObjectToPerson(item)^.SetAge(50);
    2 :
    GVL.CastHelper.ObjectToPerson(item)^.SetName('John');
ELSE
    RETURN;
END_CASE
END_METHOD

END_FUNCTION_BLOCK

// ---- POUs/List/List_I_Observer_Test.TcPOU
FUNCTION_BLOCK List_I_Observer_Test EXTENDS TcUnit.FB_TestSuite

AddItem();
Clear();
Contains();
Foreach();
GetCapacity();
GetCount();
GetItem();
IndexOfItem();
Insert();
LastIndexOfItem();
Remove();
RemoveAt();
RemoveRange();

METHOD AddItem
VAR
    propertyObserversList : List_I_Observer_;
    observerA : PropertyObserver;
    observerB : PropertyObserver;
    actualIndex1 : INT;
    actualIndex2 : INT;
    j : INT;
END_VAR
TEST('AddPropertyObserverShouldPass');
//Assign
//Act
actualIndex1 := propertyObserversList.AddItem(observerA);
actualIndex2 := propertyObserversList.AddItem(observerB);
//Assert
AssertEquals_INT(0, actualIndex1,'check add 1');
AssertEquals_INT(1, actualIndex2,'check add 2');
TEST_FINISHED();

TEST('AddToAFullListShouldReturnMinusOne');
//Assign
propertyObserversList.Clear();
FOR j:=0 TO GVL.LIST_UPPER_BOUND DO
    propertyObserversList.AddItem(observerA);
END_FOR
//Act
actualIndex1 := propertyObserversList.AddItem(observerB);
//Assert
AssertEquals_INT(-1, actualIndex1,'check overflow add');
TEST_FINISHED();
END_METHOD

METHOD Clear
VAR
    propertyObserversList1 : List_I_Observer_;
    propertyObserversList2 : List_I_Observer_;
    observer : PropertyObserver;
    expectedCount : INT := 0;
    actualCount : INT;
END_VAR
TEST('ClearAFilledListShouldPass');
//Assign
propertyObserversList1.AddItem(observer);
//Act
propertyObserversList1.Clear();
actualCount := propertyObserversList1.GetCount();
//Assert
AssertEquals(expectedCount, actualCount,'');
TEST_FINISHED();

TEST('ClearAnEmptyListShouldPass');
//Assign
expectedCount := 0;
//Act
propertyObserversList2.Clear();
actualCount := propertyObserversList2.GetCount();
//Assert
AssertEquals(expectedCount, actualCount,'');
TEST_FINISHED();
END_METHOD

METHOD Contains
VAR
    propertyObserversList : List_I_Observer_;
    observerA : PropertyObserver;
    observerB : PropertyObserver;
    observerC : PropertyObserver;
    observerD : PropertyObserver;
    observerE : PropertyObserver;
    observerF : PropertyObserver;
    observerG : PropertyObserver;
    actual : BOOL;
END_VAR
////Before All
propertyObserversList.AddItem(observerA);
propertyObserversList.AddItem(observerB);
propertyObserversList.AddItem(observerC);
propertyObserversList.AddItem(observerD);
propertyObserversList.AddItem(observerE);
propertyObserversList.AddItem(observerF);

TEST('ContainsShouldReturnTrue');
//Assign
//Act
actual := propertyObserversList.Contains(observerC);
//Assert
AssertTrue(actual,'Looking for observerC');
TEST_FINISHED();

TEST('ContainsShouldReturnFalse');
//Assign
//Act
actual := propertyObserversList.Contains(observerG);
//Assert
AssertFalse(actual,'Looking for observerG');
TEST_FINISHED();
END_METHOD

METHOD Foreach
VAR
    propertyObserversList : List_I_Observer_;
    observerA : PropertyObserver;
    observerB : PropertyObserver;
    observerC : PropertyObserver;
    observerD : PropertyObserver;
    observerE : PropertyObserver;
    action_I_Observer : Action_I_Observer_;
    actualPtPropertyObserverArray : ARRAY[0..3] OF POINTER TO PropertyObserver;
    j : INT;
END_VAR
TEST('ForeachByDoingActionOneShouldPass');
//Assign
observerA.SetCounter(101);
observerB.SetCounter(102);
observerC.SetCounter(103);
observerD.SetCounter(104);
propertyObserversList.AddItem(observerA);
propertyObserversList.AddItem(observerB);
propertyObserversList.AddItem(observerC);
propertyObserversList.AddItem(observerD);
//Act
propertyObserversList.Foreach(action_I_Observer, 1);
FOR j:=0 TO 3 DO
    __QUERYPOINTER(propertyObserversList.GetItem(j), actualPtPropertyObserverArray[j]);
END_FOR
//Assert
AssertEquals_INT(102, actualPtPropertyObserverArray[0]^.GetCounter(),'element 0 counter shuold be increment 1');
AssertEquals_INT(103, actualPtPropertyObserverArray[1]^.GetCounter(),'element 1 counter shuold be increment 1');
AssertEquals_INT(104, actualPtPropertyObserverArray[2]^.GetCounter(),'element 2 counter shuold be increment 1');
AssertEquals_INT(105, actualPtPropertyObserverArray[3]^.GetCounter(),'element 3 counter shuold be increment 1');
TEST_FINISHED();

TEST('ForeachByDoingActionTwoShouldPass');
//Assign
observerA.SetCounter(101);
observerB.SetCounter(102);
observerC.SetCounter(103);
observerD.SetCounter(104);
propertyObserversList.Clear();
propertyObserversList.AddItem(observerA);
propertyObserversList.AddItem(observerB);
propertyObserversList.AddItem(observerC);
propertyObserversList.AddItem(observerD);
//Act
propertyObserversList.Foreach(action_I_Observer, 2);
FOR j:=0 TO 3 DO
    __QUERYPOINTER(propertyObserversList.GetItem(j), actualPtPropertyObserverArray[j]);
END_FOR
//Assert
AssertEquals_INT(100, actualPtPropertyObserverArray[0]^.GetCounter(),'element 0 counter shuold be decrement 1');
AssertEquals_INT(101, actualPtPropertyObserverArray[1]^.GetCounter(),'element 1 counter shuold be decrement 1');
AssertEquals_INT(102, actualPtPropertyObserverArray[2]^.GetCounter(),'element 2 counter shuold be decrement 1');
AssertEquals_INT(103, actualPtPropertyObserverArray[3]^.GetCounter(),'element 3 counter shuold be decrement 1');
TEST_FINISHED();
END_METHOD

METHOD GetCapacity
VAR
    propertyObserversList : List_I_Observer_;
    observer : PropertyObserver;
    expectedCapacity : INT := GVL.LIST_UPPER_BOUND + 1;
    actualCapacity : INT;
END_VAR
TEST('GetCapacityShouldPass');
//Act
actualCapacity := propertyObserversList.GetCapacity();
//Assert
AssertEquals_INT(expectedCapacity, actualCapacity,'Get capacity at the begining');
TEST_FINISHED();

TEST('GetCapacityShouldPassWithSameValue');
//Assign
propertyObserversList.AddItem(observer);
//Act
actualCapacity := propertyObserversList.GetCapacity();
//Assert
AssertEquals(expectedCapacity, actualCapacity,'Get capacity after adding an observer');
TEST_FINISHED();
END_METHOD

METHOD GetCount
VAR
    propertyObserversList : List_I_Observer_;
    observer : PropertyObserver;
    expectedCount : INT := 0;
    actualCount : INT;
END_VAR
TEST('GetCountShouldReturnZero');
//Act
actualCount := propertyObserversList.GetCount();
//Assert
AssertEquals_INT(expectedCount, actualCount,'Get count at the begining');
TEST_FINISHED();

TEST('GetCountShouldReturnOne');
//Assign
propertyObserversList.AddItem(observer);
expectedCount := 1;
//Act
actualCount := propertyObserversList.GetCount();
//Assert
AssertEquals(expectedCount, actualCount,'Get count after adding an observer');
TEST_FINISHED();
END_METHOD

METHOD GetItem
VAR
    propertyObserversList : List_I_Observer_;
    expectedObserverA : PropertyObserver;
    expectedObserverB : PropertyObserver;
    actualObserver : I_Observer;
    actualPropertyObserverA : POINTER TO PropertyObserver;
    actualPropertyObserverB : POINTER TO PropertyObserver;
    expectedIndex : INT := 0;
    actualIndex : INT;
END_VAR
TEST('GetPropertyObserverShouldPass');
//Assign
expectedObserverA.SetCounter(101);
expectedObserverB.SetCounter(102);
propertyObserversList.AddItem(expectedObserverA);
propertyObserversList.AddItem(expectedObserverB);
//Act
actualObserver := propertyObserversList.GetItem(0);
__QUERYPOINTER(actualObserver, actualPropertyObserverA);
actualObserver := propertyObserversList.GetItem(1);
__QUERYPOINTER(actualObserver, actualPropertyObserverB);
//Assert
AssertTrue(actualPropertyObserverA^.Equals(expectedObserverA),'check A');
AssertTrue(actualPropertyObserverB^.Equals(expectedObserverB),'check B');
TEST_FINISHED();
END_METHOD

METHOD IndexOfItem
VAR
    propertyObserversList : List_I_Observer_;
    observerA : PropertyObserver;
    observerB : PropertyObserver;
    observerC : PropertyObserver;
    observerD : PropertyObserver;
    observerE : PropertyObserver;
    observerF : PropertyObserver;
    observerG : PropertyObserver;
    actualIndex : INT;
    expectedIndex : INT := 3;
END_VAR
//Before All
propertyObserversList.AddItem(observerA);
propertyObserversList.AddItem(observerB);
propertyObserversList.AddItem(observerC);
propertyObserversList.AddItem(observerD);
propertyObserversList.AddItem(observerE);
propertyObserversList.AddItem(observerF);

TEST('IndexOfItemShouldReturnTheIndex');
//Assign
//Act
actualIndex := propertyObserversList.IndexOfItem(observerD);
//Assert
AssertEquals(expectedIndex, actualIndex, 'return the index of observerD');
TEST_FINISHED();

TEST('IndexOfItemShouldReturnMinusOne');
//Assign
//Act
actualIndex := propertyObserversList.IndexOfItem(observerG);
//Assert
expectedIndex := -1;
AssertEquals(expectedIndex, actualIndex, 'return the index of observerG');
TEST_FINISHED();
END_METHOD

METHOD Insert
VAR
    propertyObserversList : List_I_Observer_;
    observerA : PropertyObserver;
    observerB : PropertyObserver;
    observerC : PropertyObserver;
    observerD : PropertyObserver;
    actualPtPropertyObserverArray : ARRAY[0..3] OF POINTER TO PropertyObserver;
    expected : INT := 2;
    actual : INT;
    j : INT;
END_VAR
//Before All
observerA.SetCounter(101);
observerB.SetCounter(102);
observerC.SetCounter(103);
observerD.SetCounter(104);

TEST('InsertShouldPassAndReturnTheLastIndex');
//Assign
propertyObserversList.AddItem(observerA);
propertyObserversList.AddItem(observerB);
propertyObserversList.AddItem(observerC);
//Act
actual := propertyObserversList.Insert(2, observerD);
FOR j:=0 TO 3 DO
    __QUERYPOINTER(propertyObserversList.GetItem(j), actualPtPropertyObserverArray[j]);
END_FOR
//Assert
AssertEquals(expected, actual, 'check result');
AssertEquals_INT(4, propertyObserversList.GetCount(),'check list count');
AssertTrue(actualPtPropertyObserverArray[0]^.Equals(observerA),'check element 0');
AssertTrue(actualPtPropertyObserverArray[1]^.Equals(observerB),'check element 1');
AssertTrue(actualPtPropertyObserverArray[2]^.Equals(observerD),'check element 2');
AssertTrue(actualPtPropertyObserverArray[3]^.Equals(observerC),'check element 3');
TEST_FINISHED();

TEST('InsertShouldPassEvenByIndexHigherThanListCurrentLastIndexAndReturnTheLastIndex');
//Assign
propertyObserversList.Clear();
propertyObserversList.AddItem(observerA);
propertyObserversList.AddItem(observerB);
propertyObserversList.AddItem(observerC);
expected := 3;
//Act
actual := propertyObserversList.Insert(7, observerD);
FOR j:=0 TO 3 DO
    __QUERYPOINTER(propertyObserversList.GetItem(j), actualPtPropertyObserverArray[j]);
END_FOR
//Assert
AssertEquals(expected, actual, 'check result');
AssertEquals_INT(4, propertyObserversList.GetCount(),'check list count');
AssertTrue(actualPtPropertyObserverArray[0]^.Equals(observerA),'check element 0');
AssertTrue(actualPtPropertyObserverArray[1]^.Equals(observerB),'check element 1');
AssertTrue(actualPtPropertyObserverArray[2]^.Equals(observerC),'check element 2');
AssertTrue(actualPtPropertyObserverArray[3]^.Equals(observerD),'check element 3');
TEST_FINISHED();

TEST('InsertShouldPassEvenByIndexHigherThanListUpperBoundAndReturnTheLastIndex');
//Assign
propertyObserversList.Clear();
propertyObserversList.AddItem(observerA);
propertyObserversList.AddItem(observerB);
propertyObserversList.AddItem(observerC);
expected := 3;
//Act
actual := propertyObserversList.Insert(GVL.LIST_UPPER_BOUND + 1, observerD);
FOR j:=0 TO 3 DO
    __QUERYPOINTER(propertyObserversList.GetItem(j), actualPtPropertyObserverArray[j]);
END_FOR
//Assert
AssertEquals(expected, actual, 'check result');
AssertEquals_INT(4, propertyObserversList.GetCount(),'check list count');
AssertTrue(actualPtPropertyObserverArray[0]^.Equals(observerA),'check element 0');
AssertTrue(actualPtPropertyObserverArray[1]^.Equals(observerB),'check element 1');
AssertTrue(actualPtPropertyObserverArray[2]^.Equals(observerC),'check element 2');
AssertTrue(actualPtPropertyObserverArray[3]^.Equals(observerD),'check element 3');
TEST_FINISHED();

TEST('InsertShouldFailByMinusIndexAndReturnMinusOne');
//Assign
propertyObserversList.Clear();
propertyObserversList.AddItem(observerA);
propertyObserversList.AddItem(observerB);
propertyObserversList.AddItem(observerC);
expected := -1;
//Act
actual := propertyObserversList.Insert(-1, observerD);
//Assert
AssertEquals(expected, actual, 'check result');
AssertEquals_INT(3, propertyObserversList.GetCount(),'check list count');
TEST_FINISHED();
END_METHOD

METHOD LastIndexOfItem
VAR
    propertyObserversList : List_I_Observer_;
    observerA : PropertyObserver;
    observerB : PropertyObserver;
    observerC : PropertyObserver;
    observerD : PropertyObserver;
    observerE : PropertyObserver;
    observerF : PropertyObserver;
    observerG : PropertyObserver;
    actualIndex : INT;
    expectedIndex : INT := 5;
END_VAR
//Before All
propertyObserversList.AddItem(observerA);
propertyObserversList.AddItem(observerB);
propertyObserversList.AddItem(observerC);
propertyObserversList.AddItem(observerD);
propertyObserversList.AddItem(observerE);
propertyObserversList.AddItem(observerD);
propertyObserversList.AddItem(observerF);

TEST('LastIndexOfItemShouldReturnTheIndex');
//Assign
//Act
actualIndex := propertyObserversList.LastIndexOfItem(observerD);
//Assert
AssertEquals(expectedIndex, actualIndex, 'return the last index of observerD');
TEST_FINISHED();

TEST('LastIndexOfItemShouldReturnMinusOne');
//Assign
//Act
actualIndex := propertyObserversList.LastIndexOfItem(observerG);
//Assert
expectedIndex := -1;
AssertEquals(expectedIndex, actualIndex, 'return the last index of observerG');
TEST_FINISHED();
END_METHOD

METHOD Remove
VAR
    propertyObserversList : List_I_Observer_;
    observerA : PropertyObserver;
    observerB : PropertyObserver;
    observerC : PropertyObserver;
    observerD : PropertyObserver;
    actualPtPropertyObserverArray : ARRAY[0..3] OF POINTER TO PropertyObserver;
    expectedCount : INT := 3;
    actualCount : INT;
    actual : BOOL;
    j : INT;
END_VAR
//Before All
observerA.SetCounter(101);
observerB.SetCounter(102);
observerC.SetCounter(103);
observerD.SetCounter(104);
propertyObserversList.AddItem(observerA);
propertyObserversList.AddItem(observerB);
propertyObserversList.AddItem(observerC);
propertyObserversList.AddItem(observerD);

TEST('RemoveShouldPassAndReturnTrue');
//Assign
//Act
actual := propertyObserversList.Remove(observerC);
actualCount := propertyObserversList.GetCount();
FOR j:=0 TO 3 DO
    __QUERYPOINTER(propertyObserversList.GetItem(j), actualPtPropertyObserverArray[j]);
END_FOR
//Assert
AssertTrue(actual,'check result of remove');
AssertEquals(expectedCount, actualCount,'check list count');
AssertTrue(actualPtPropertyObserverArray[0]^.Equals(observerA),'check list element 0');
AssertTrue(actualPtPropertyObserverArray[1]^.Equals(observerB),'check list element 1');
AssertTrue(actualPtPropertyObserverArray[2]^.Equals(observerD),'check list element 2');
TEST_FINISHED();

TEST('RemoveShouldFailAndReturnFalse');
//Assign
//Act
actual := propertyObserversList.Remove(observerC);
actualCount := propertyObserversList.GetCount();
FOR j:=0 TO 3 DO
    __QUERYPOINTER(propertyObserversList.GetItem(j), actualPtPropertyObserverArray[j]);
END_FOR
//Assert
AssertFalse(actual,'check result of remove');
AssertEquals(expectedCount, actualCount,'check list count');
AssertTrue(actualPtPropertyObserverArray[0]^.Equals(observerA),'check list element 0');
AssertTrue(actualPtPropertyObserverArray[1]^.Equals(observerB),'check list element 1');
AssertTrue(actualPtPropertyObserverArray[2]^.Equals(observerD),'check list element 2');
TEST_FINISHED();
END_METHOD

METHOD RemoveAt
VAR
    propertyObserversList : List_I_Observer_;
    observerA : PropertyObserver;
    observerB : PropertyObserver;
    observerC : PropertyObserver;
    observerD : PropertyObserver;
    actualPtPropertyObserverArray : ARRAY[0..3] OF POINTER TO PropertyObserver;
    expectedCount : INT := 3;
    actualCount : INT;
    actual : BOOL;
    j : INT;
END_VAR
observerA.SetCounter(101);
observerB.SetCounter(102);
observerC.SetCounter(103);
observerD.SetCounter(104);

